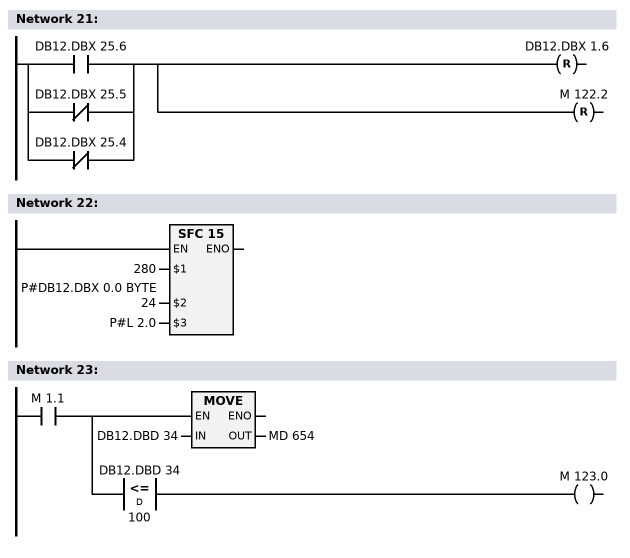
NETWORK
TITLE =
      O     DB12.DBX 25.6;
      ON    DB12.DBX 25.5;
      ON    DB12.DBX 25.4;
      R     DB12.DBX 1.6;
      R     M 122.2;
NETWORK
TITLE =
      CALL  SFC 15 (
           $1                       := 280,
           $2                       := P#DB12.DBX 0.0 BYTE 24,
           $3                       := P#L 2.0);
      NOP   0;
NETWORK
TITLE =
      A     M 1.1;
      =     L 20.0;
      A     L 20.0;
      JNB   M019;
      L     DB12.DBD 34;
      T     MD 654;
M019: NOP   0;
      A     L 20.0;
      A(;
      L     DB12.DBD 34;
      L     100;
      <=D;
      );
      =     M 123.0;
END_FUNCTION

FUNCTION FC 50 : VOID
VERSION : 0.1
BEGIN
// (block stored without names or comments; labels and parameter names are numbered)
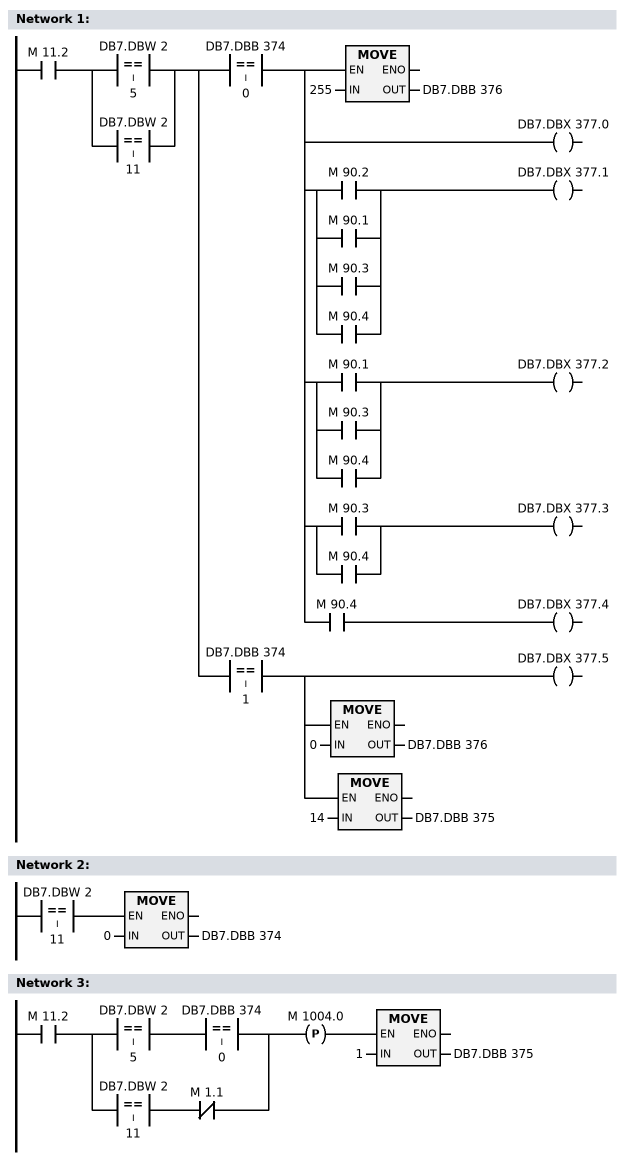
NETWORK
TITLE =
      A     M 11.2;
      A(;
      O(;
      L     DB7.DBW 2;
      L     5;
      ==I;
      );
      O(;
      L     DB7.DBW 2;
      L     11;
      ==I;
      );
      );
      =     L 8.0;
      A     L 8.0;
      A(;
      L     DB7.DBB 374;
      L     0;
      ==I;
      );
      =     L 8.1;
      A     L 8.1;
      JNB   M001;
      L     255;
      T     DB7.DBB 376;
M001: NOP   0;
      A     L 8.1;
      BLD   102;
      =     DB7.DBX 377.0;
      A     L 8.1;
      A(;
      O     M 90.2;
      O     M 90.1;
      O     M 90.3;
      O     M 90.4;
      );
      =     DB7.DBX 377.1;
      A     L 8.1;
      A(;
      O     M 90.1;
      O     M 90.3;
      O     M 90.4;
      );
      =     DB7.DBX 377.2;
      A     L 8.1;
      A(;
      O     M 90.3;
      O     M 90.4;
      );
      =     DB7.DBX 377.3;
      A     L 8.1;
      A     M 90.4;
      =     DB7.DBX 377.4;
      A     L 8.0;
      A(;
      L     DB7.DBB 374;
      L     1;
      ==I;
      );
      =     L 8.1;
      A     L 8.1;
      BLD   102;
      =     DB7.DBX 377.5;
      A     L 8.1;
      JNB   M002;
      L     0;
      T     DB7.DBB 376;
M002: NOP   0;
      A     L 8.1;
      JNB   M003;
      L     14;
      T     DB7.DBB 375;
M003: NOP   0;
NETWORK
TITLE =
      A(;
      L     DB7.DBW 2;
      L     11;
      ==I;
      );
      JNB   M004;
      L     0;
      T     DB7.DBB 374;
M004: NOP   0;
NETWORK
TITLE =
      A     M 11.2;
      A(;
      A(;
      L     DB7.DBW 2;
      L     5;
      ==I;
      );
      A(;
      L     DB7.DBB 374;
      L     0;
      ==I;
      );
      O;
      A(;
      L     DB7.DBW 2;
      L     11;
      ==I;
      );
      AN    M 1.1;
      );
      FP    M 1004.0;
      JNB   M005;
      L     1;
      T     DB7.DBB 375;
M005: NOP   0;
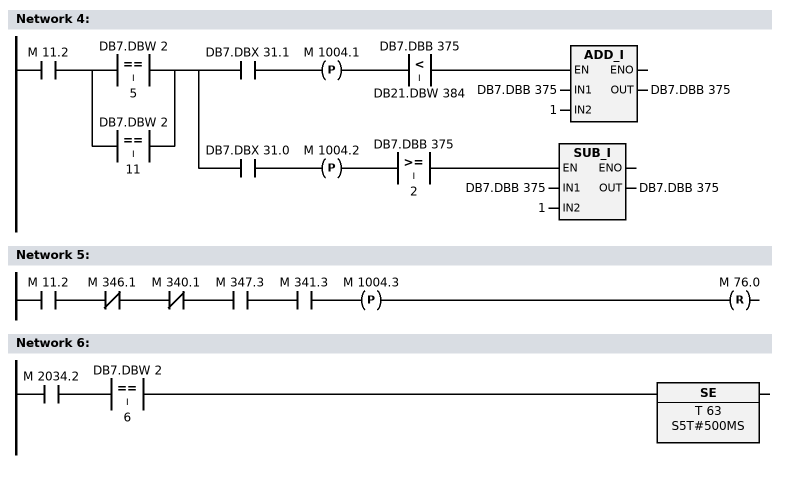
NETWORK
TITLE =
      A     M 11.2;
      A(;
      O(;
      L     DB7.DBW 2;
      L     5;
      ==I;
      );
      O(;
      L     DB7.DBW 2;
      L     11;
      ==I;
      );
      );
      =     L 8.0;
      A     L 8.0;
      A     DB7.DBX 31.1;
      FP    M 1004.1;
      A(;
      L     DB7.DBB 375;
      L     DB21.DBW 384;
      <I;
      );
      JNB   M006;
      L     DB7.DBB 375;
      L     1;
      +I;
      T     DB7.DBB 375;
M006: NOP   0;
      A     L 8.0;
      A     DB7.DBX 31.0;
      FP    M 1004.2;
      A(;
      L     DB7.DBB 375;
      L     2;
      >=I;
      );
      JNB   M007;
      L     DB7.DBB 375;
      L     1;
      -I;
      T     DB7.DBB 375;
M007: NOP   0;
NETWORK
TITLE =
      A     M 11.2;
      AN    M 346.1;
      AN    M 340.1;
      A     M 347.3;
      A     M 341.3;
      FP    M 1004.3;
      R     M 76.0;
NETWORK
TITLE =
      A     M 2034.2;
      A(;
      L     DB7.DBW 2;
      L     6;
      ==I;
      );
      L     S5T#500MS;
      SE    T 63;
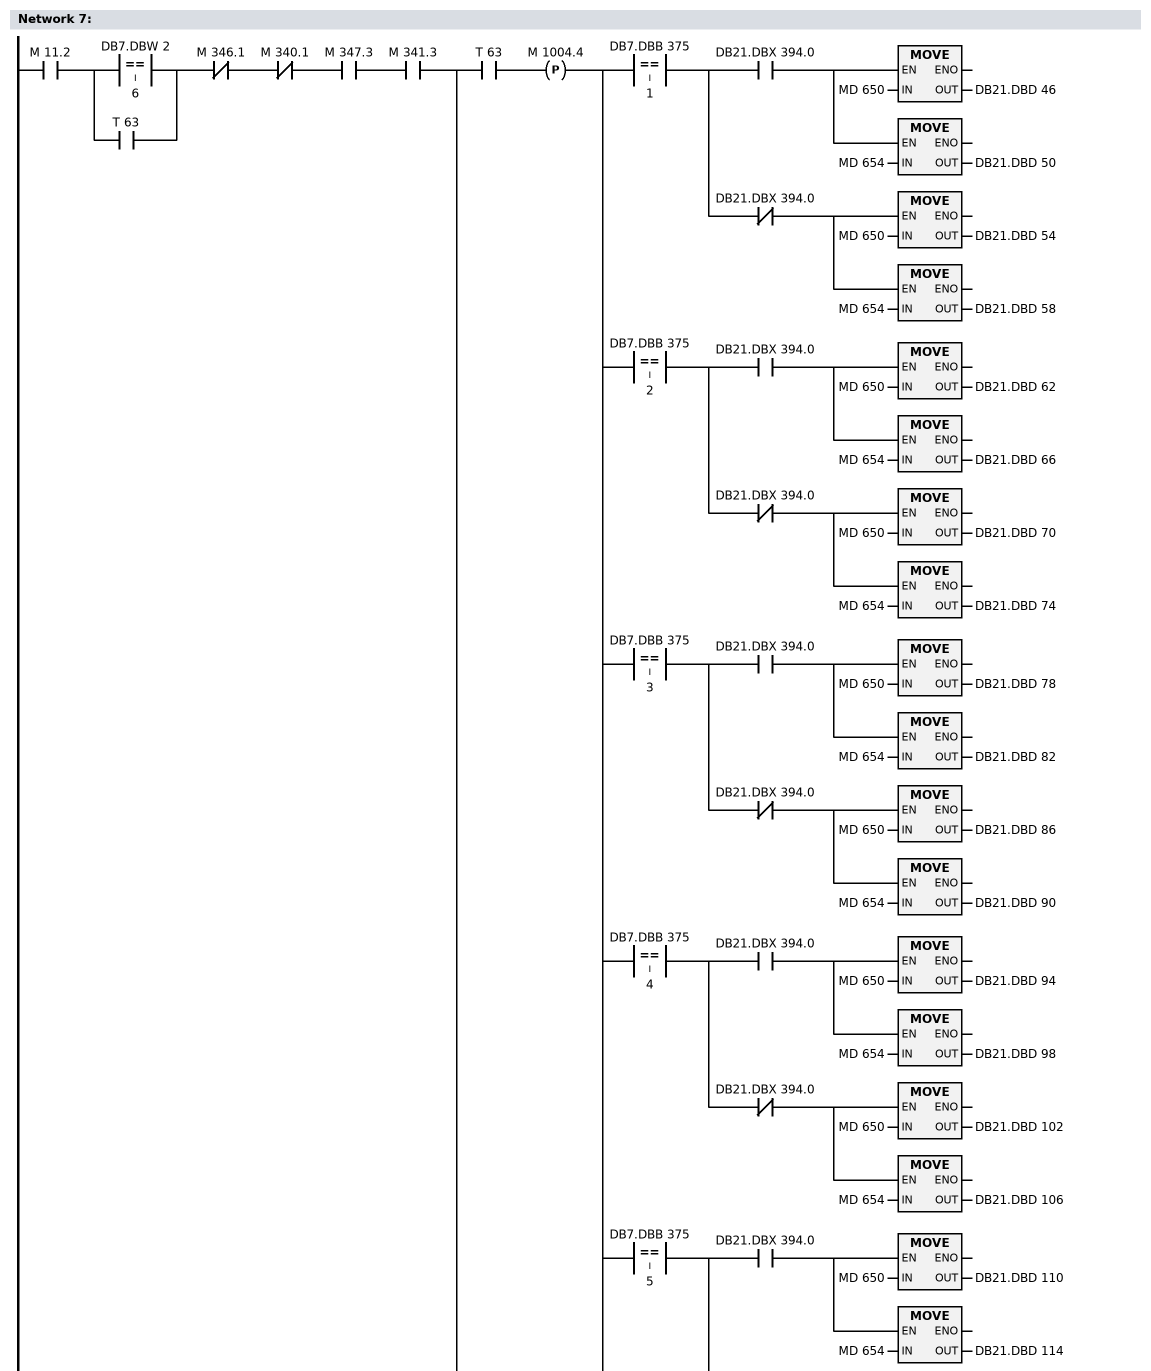
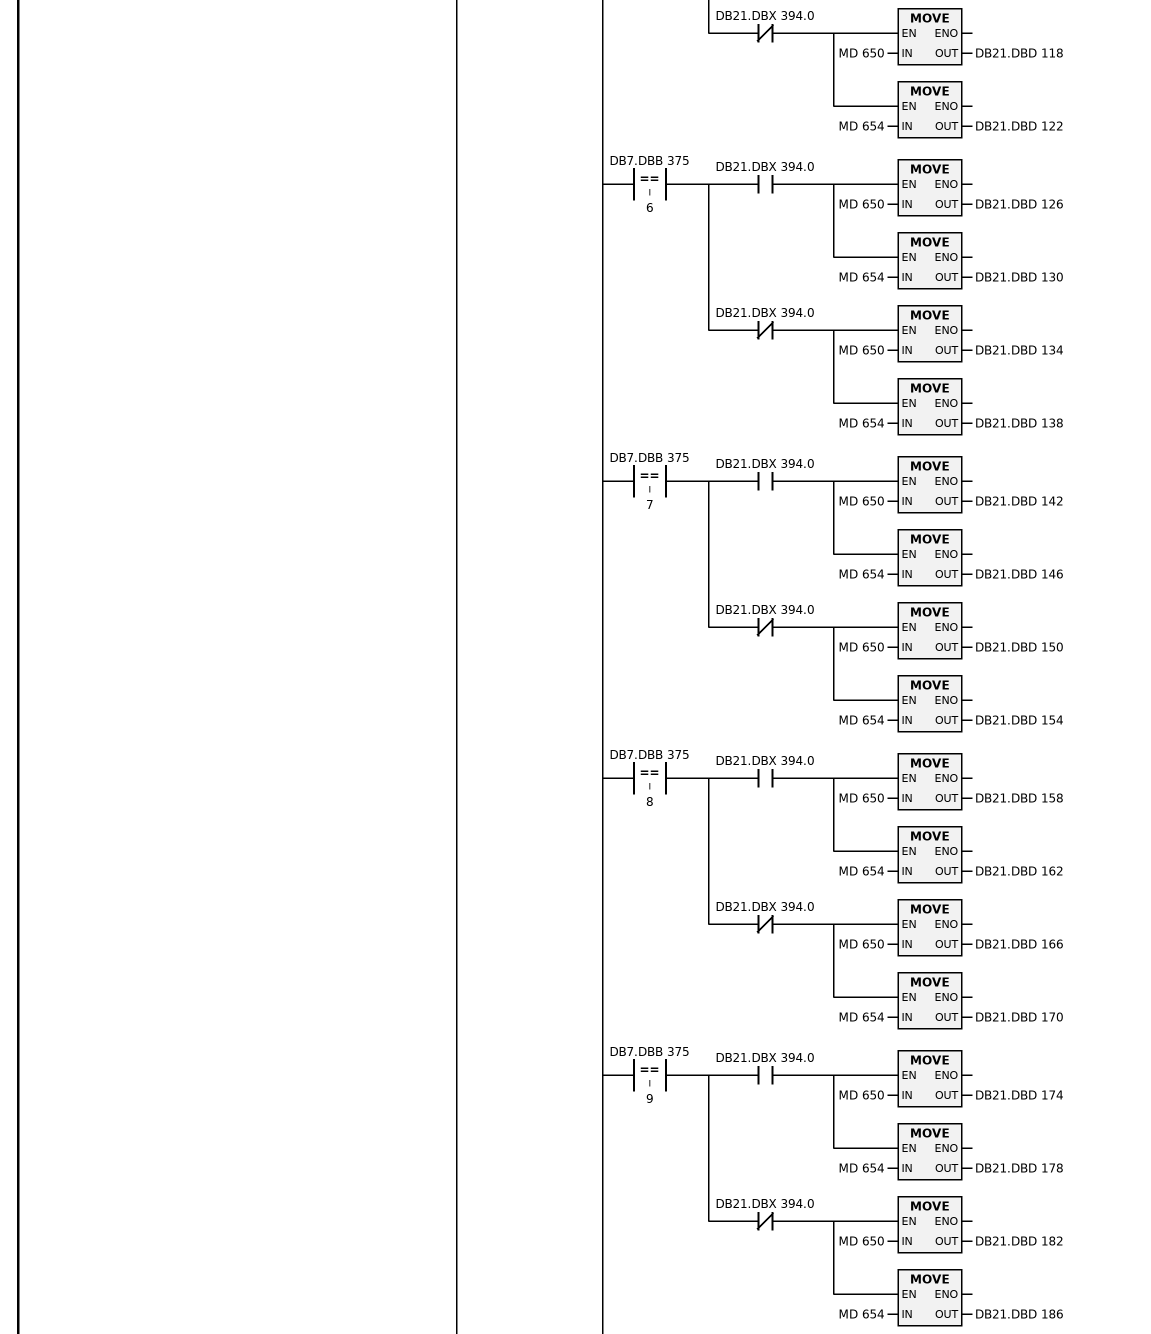
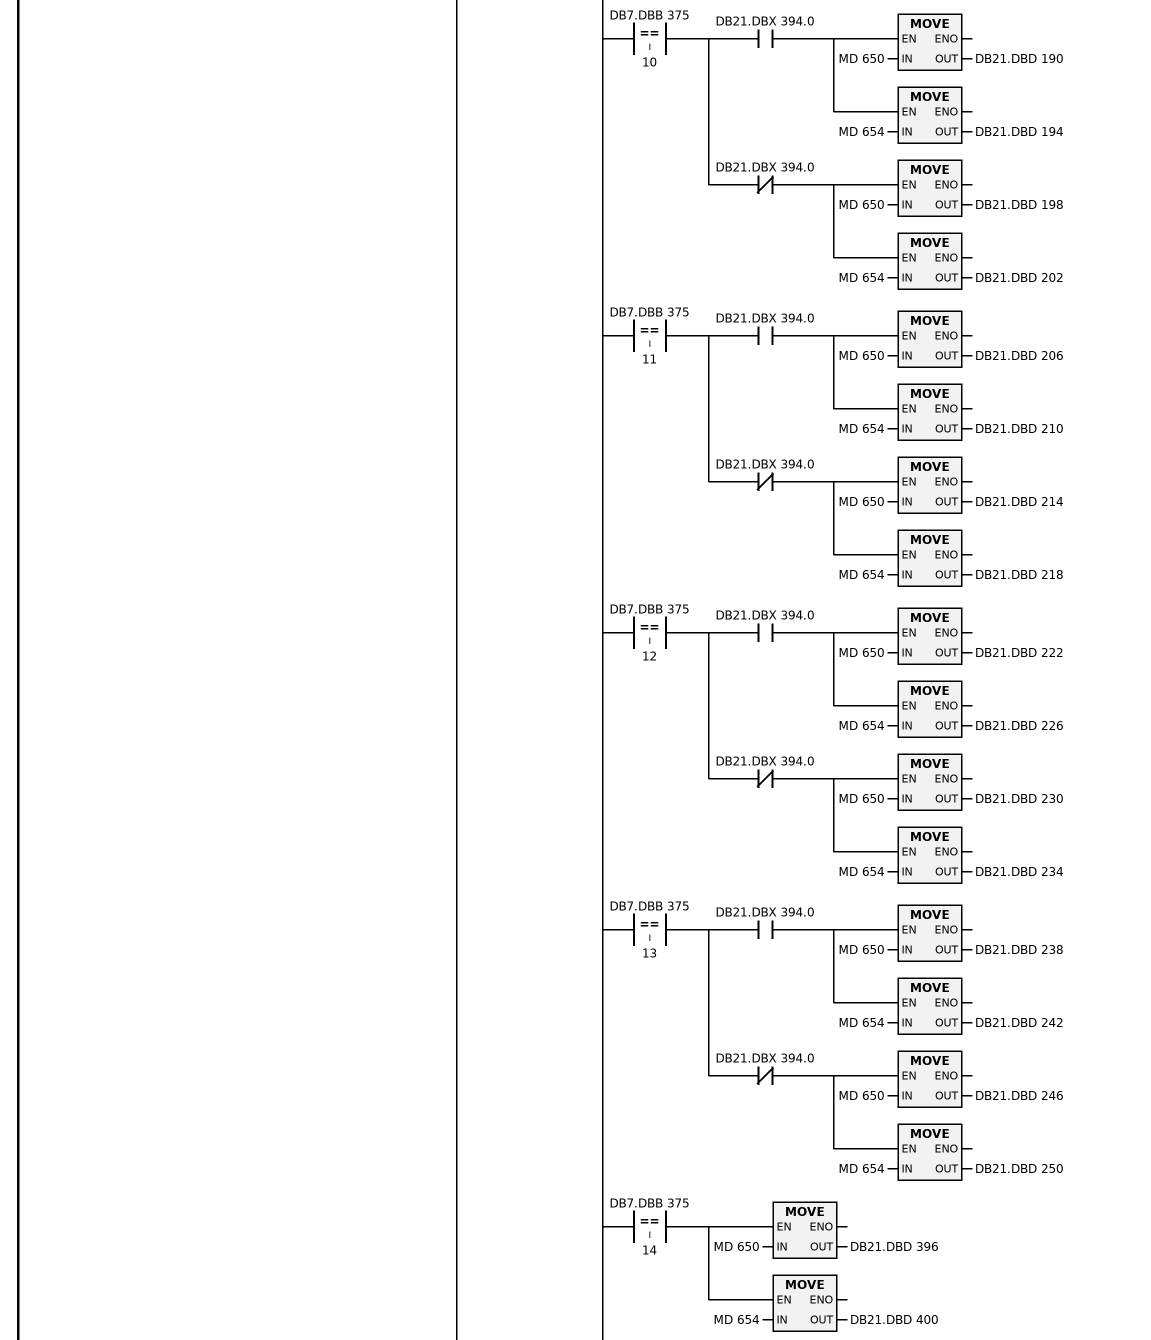
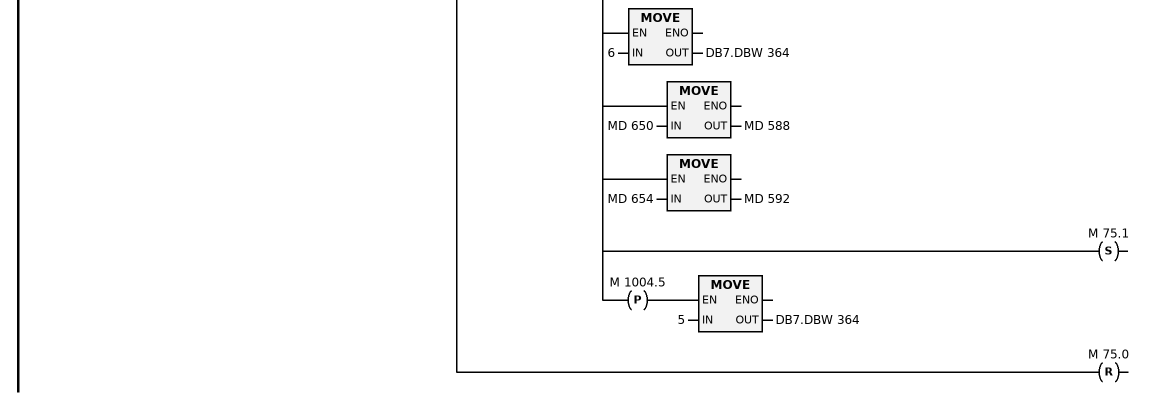
NETWORK
TITLE =
      A     M 11.2;
      A(;
      O(;
      L     DB7.DBW 2;
      L     6;
      ==I;
      );
      O     T 63;
      );
      AN    M 346.1;
      AN    M 340.1;
      A     M 347.3;
      A     M 341.3;
      =     L 8.0;
      A     L 8.0;
      A     T 63;
      FP    M 1004.4;
      =     L 8.1;
      A     L 8.1;
      A(;
      L     DB7.DBB 375;
      L     1;
      ==I;
      );
      =     L 8.2;
      A     L 8.2;
      A     DB21.DBX 394.0;
      =     L 8.3;
      A     L 8.3;
      JNB   M008;
      L     MD 650;
      T     DB21.DBD 46;
M008: NOP   0;
      A     L 8.3;
      JNB   M009;
      L     MD 654;
      T     DB21.DBD 50;
M009: NOP   0;
      A     L 8.2;
      AN    DB21.DBX 394.0;
      =     L 8.3;
      A     L 8.3;
      JNB   M010;
      L     MD 650;
      T     DB21.DBD 54;
M010: NOP   0;
      A     L 8.3;
      JNB   M011;
      L     MD 654;
      T     DB21.DBD 58;
M011: NOP   0;
      A     L 8.1;
      A(;
      L     DB7.DBB 375;
      L     2;
      ==I;
      );
      =     L 8.2;
      A     L 8.2;
      A     DB21.DBX 394.0;
      =     L 8.3;
      A     L 8.3;
      JNB   M012;
      L     MD 650;
      T     DB21.DBD 62;
M012: NOP   0;
      A     L 8.3;
      JNB   M013;
      L     MD 654;
      T     DB21.DBD 66;
M013: NOP   0;
      A     L 8.2;
      AN    DB21.DBX 394.0;
      =     L 8.3;
      A     L 8.3;
      JNB   M014;
      L     MD 650;
      T     DB21.DBD 70;
M014: NOP   0;
      A     L 8.3;
      JNB   M015;
      L     MD 654;
      T     DB21.DBD 74;
M015: NOP   0;
      A     L 8.1;
      A(;
      L     DB7.DBB 375;
      L     3;
      ==I;
      );
      =     L 8.2;
      A     L 8.2;
      A     DB21.DBX 394.0;
      =     L 8.3;
      A     L 8.3;
      JNB   M016;
      L     MD 650;
      T     DB21.DBD 78;
M016: NOP   0;
      A     L 8.3;
      JNB   M017;
      L     MD 654;
      T     DB21.DBD 82;
M017: NOP   0;
      A     L 8.2;
      AN    DB21.DBX 394.0;
      =     L 8.3;
      A     L 8.3;
      JNB   M018;
      L     MD 650;
      T     DB21.DBD 86;
M018: NOP   0;
      A     L 8.3;
      JNB   M019;
      L     MD 654;
      T     DB21.DBD 90;
M019: NOP   0;
      A     L 8.1;
      A(;
      L     DB7.DBB 375;
      L     4;
      ==I;
      );
      =     L 8.2;
      A     L 8.2;
      A     DB21.DBX 394.0;
      =     L 8.3;
      A     L 8.3;
      JNB   M020;
      L     MD 650;
      T     DB21.DBD 94;
M020: NOP   0;
      A     L 8.3;
      JNB   M021;
      L     MD 654;
      T     DB21.DBD 98;
M021: NOP   0;
      A     L 8.2;
      AN    DB21.DBX 394.0;
      =     L 8.3;
      A     L 8.3;
      JNB   M022;
      L     MD 650;
      T     DB21.DBD 102;
M022: NOP   0;
      A     L 8.3;
      JNB   M023;
      L     MD 654;
      T     DB21.DBD 106;
M023: NOP   0;
      A     L 8.1;
      A(;
      L     DB7.DBB 375;
      L     5;
      ==I;
      );
      =     L 8.2;
      A     L 8.2;
      A     DB21.DBX 394.0;
      =     L 8.3;
      A     L 8.3;
      JNB   M024;
      L     MD 650;
      T     DB21.DBD 110;
M024: NOP   0;
      A     L 8.3;
      JNB   M025;
      L     MD 654;
      T     DB21.DBD 114;
M025: NOP   0;
      A     L 8.2;
      AN    DB21.DBX 394.0;
      =     L 8.3;
      A     L 8.3;
      JNB   M026;
      L     MD 650;
      T     DB21.DBD 118;
M026: NOP   0;
      A     L 8.3;
      JNB   M027;
      L     MD 654;
      T     DB21.DBD 122;
M027: NOP   0;
      A     L 8.1;
      A(;
      L     DB7.DBB 375;
      L     6;
      ==I;
      );
      =     L 8.2;
      A     L 8.2;
      A     DB21.DBX 394.0;
      =     L 8.3;
      A     L 8.3;
      JNB   M028;
      L     MD 650;
      T     DB21.DBD 126;
M028: NOP   0;
      A     L 8.3;
      JNB   M029;
      L     MD 654;
      T     DB21.DBD 130;
M029: NOP   0;
      A     L 8.2;
      AN    DB21.DBX 394.0;
      =     L 8.3;
      A     L 8.3;
      JNB   M030;
      L     MD 650;
      T     DB21.DBD 134;
M030: NOP   0;
      A     L 8.3;
      JNB   M031;
      L     MD 654;
      T     DB21.DBD 138;
M031: NOP   0;
      A     L 8.1;
      A(;
      L     DB7.DBB 375;
      L     7;
      ==I;
      );
      =     L 8.2;
      A     L 8.2;
      A     DB21.DBX 394.0;
      =     L 8.3;
      A     L 8.3;
      JNB   M032;
      L     MD 650;
      T     DB21.DBD 142;
M032: NOP   0;
      A     L 8.3;
      JNB   M033;
      L     MD 654;
      T     DB21.DBD 146;
M033: NOP   0;
      A     L 8.2;
      AN    DB21.DBX 394.0;
      =     L 8.3;
      A     L 8.3;
      JNB   M034;
      L     MD 650;
      T     DB21.DBD 150;
M034: NOP   0;
      A     L 8.3;
      JNB   M035;
      L     MD 654;
      T     DB21.DBD 154;
M035: NOP   0;
      A     L 8.1;
      A(;
      L     DB7.DBB 375;
      L     8;
      ==I;
      );
      =     L 8.2;
      A     L 8.2;
      A     DB21.DBX 394.0;
      =     L 8.3;
      A     L 8.3;
      JNB   M036;
      L     MD 650;
      T     DB21.DBD 158;
M036: NOP   0;
      A     L 8.3;
      JNB   M037;
      L     MD 654;
      T     DB21.DBD 162;
M037: NOP   0;
      A     L 8.2;
      AN    DB21.DBX 394.0;
      =     L 8.3;
      A     L 8.3;
      JNB   M038;
      L     MD 650;
      T     DB21.DBD 166;
M038: NOP   0;
      A     L 8.3;
      JNB   M039;
      L     MD 654;
      T     DB21.DBD 170;
M039: NOP   0;
      A     L 8.1;
      A(;
      L     DB7.DBB 375;
      L     9;
      ==I;
      );
      =     L 8.2;
      A     L 8.2;
      A     DB21.DBX 394.0;
      =     L 8.3;
      A     L 8.3;
      JNB   M040;
      L     MD 650;
      T     DB21.DBD 174;
M040: NOP   0;
      A     L 8.3;
      JNB   M041;
      L     MD 654;
      T     DB21.DBD 178;
M041: NOP   0;
      A     L 8.2;
      AN    DB21.DBX 394.0;
      =     L 8.3;
      A     L 8.3;
      JNB   M042;
      L     MD 650;
      T     DB21.DBD 182;
M042: NOP   0;
      A     L 8.3;
      JNB   M043;
      L     MD 654;
      T     DB21.DBD 186;
M043: NOP   0;
      A     L 8.1;
      A(;
      L     DB7.DBB 375;
      L     10;
      ==I;
      );
      =     L 8.2;
      A     L 8.2;
      A     DB21.DBX 394.0;
      =     L 8.3;
      A     L 8.3;
      JNB   M044;
      L     MD 650;
      T     DB21.DBD 190;
M044: NOP   0;
      A     L 8.3;
      JNB   M045;
      L     MD 654;
      T     DB21.DBD 194;
M045: NOP   0;
      A     L 8.2;
      AN    DB21.DBX 394.0;
      =     L 8.3;
      A     L 8.3;
      JNB   M046;
      L     MD 650;
      T     DB21.DBD 198;
M046: NOP   0;
      A     L 8.3;
      JNB   M047;
      L     MD 654;
      T     DB21.DBD 202;
M047: NOP   0;
      A     L 8.1;
      A(;
      L     DB7.DBB 375;
      L     11;
      ==I;
      );
      =     L 8.2;
      A     L 8.2;
      A     DB21.DBX 394.0;
      =     L 8.3;
      A     L 8.3;
      JNB   M048;
      L     MD 650;
      T     DB21.DBD 206;
M048: NOP   0;
      A     L 8.3;
      JNB   M049;
      L     MD 654;
      T     DB21.DBD 210;
M049: NOP   0;
      A     L 8.2;
      AN    DB21.DBX 394.0;
      =     L 8.3;
      A     L 8.3;
      JNB   M050;
      L     MD 650;
      T     DB21.DBD 214;
M050: NOP   0;
      A     L 8.3;
      JNB   M051;
      L     MD 654;
      T     DB21.DBD 218;
M051: NOP   0;
      A     L 8.1;
      A(;
      L     DB7.DBB 375;
      L     12;
      ==I;
      );
      =     L 8.2;
      A     L 8.2;
      A     DB21.DBX 394.0;
      =     L 8.3;
      A     L 8.3;
      JNB   M052;
      L     MD 650;
      T     DB21.DBD 222;
M052: NOP   0;
      A     L 8.3;
      JNB   M053;
      L     MD 654;
      T     DB21.DBD 226;
M053: NOP   0;
      A     L 8.2;
      AN    DB21.DBX 394.0;
      =     L 8.3;
      A     L 8.3;
      JNB   M054;
      L     MD 650;
      T     DB21.DBD 230;
M054: NOP   0;
      A     L 8.3;
      JNB   M055;
      L     MD 654;
      T     DB21.DBD 234;
M055: NOP   0;
      A     L 8.1;
      A(;
      L     DB7.DBB 375;
      L     13;
      ==I;
      );
      =     L 8.2;
      A     L 8.2;
      A     DB21.DBX 394.0;
      =     L 8.3;
      A     L 8.3;
      JNB   M056;
      L     MD 650;
      T     DB21.DBD 238;
M056: NOP   0;
      A     L 8.3;
      JNB   M057;
      L     MD 654;
      T     DB21.DBD 242;
M057: NOP   0;
      A     L 8.2;
      AN    DB21.DBX 394.0;
      =     L 8.3;
      A     L 8.3;
      JNB   M058;
      L     MD 650;
      T     DB21.DBD 246;
M058: NOP   0;
      A     L 8.3;
      JNB   M059;
      L     MD 654;
      T     DB21.DBD 250;
M059: NOP   0;
      A     L 8.1;
      A(;
      L     DB7.DBB 375;
      L     14;
      ==I;
      );
      =     L 8.2;
      A     L 8.2;
      JNB   M060;
      L     MD 650;
      T     DB21.DBD 396;
M060: NOP   0;
      A     L 8.2;
      JNB   M061;
      L     MD 654;
      T     DB21.DBD 400;
M061: NOP   0;
      A     L 8.1;
      JNB   M062;
      L     6;
      T     DB7.DBW 364;
M062: NOP   0;
      A     L 8.1;
      JNB   M063;
      L     MD 650;
      T     MD 588;
M063: NOP   0;
      A     L 8.1;
      JNB   M064;
      L     MD 654;
      T     MD 592;
M064: NOP   0;
      A     L 8.1;
      BLD   102;
      S     M 75.1;
      A     L 8.1;
      FP    M 1004.5;
      JNB   M065;
      L     5;
      T     DB7.DBW 364;
M065: NOP   0;
      A     L 8.0;
      BLD   102;
      R     M 75.0;
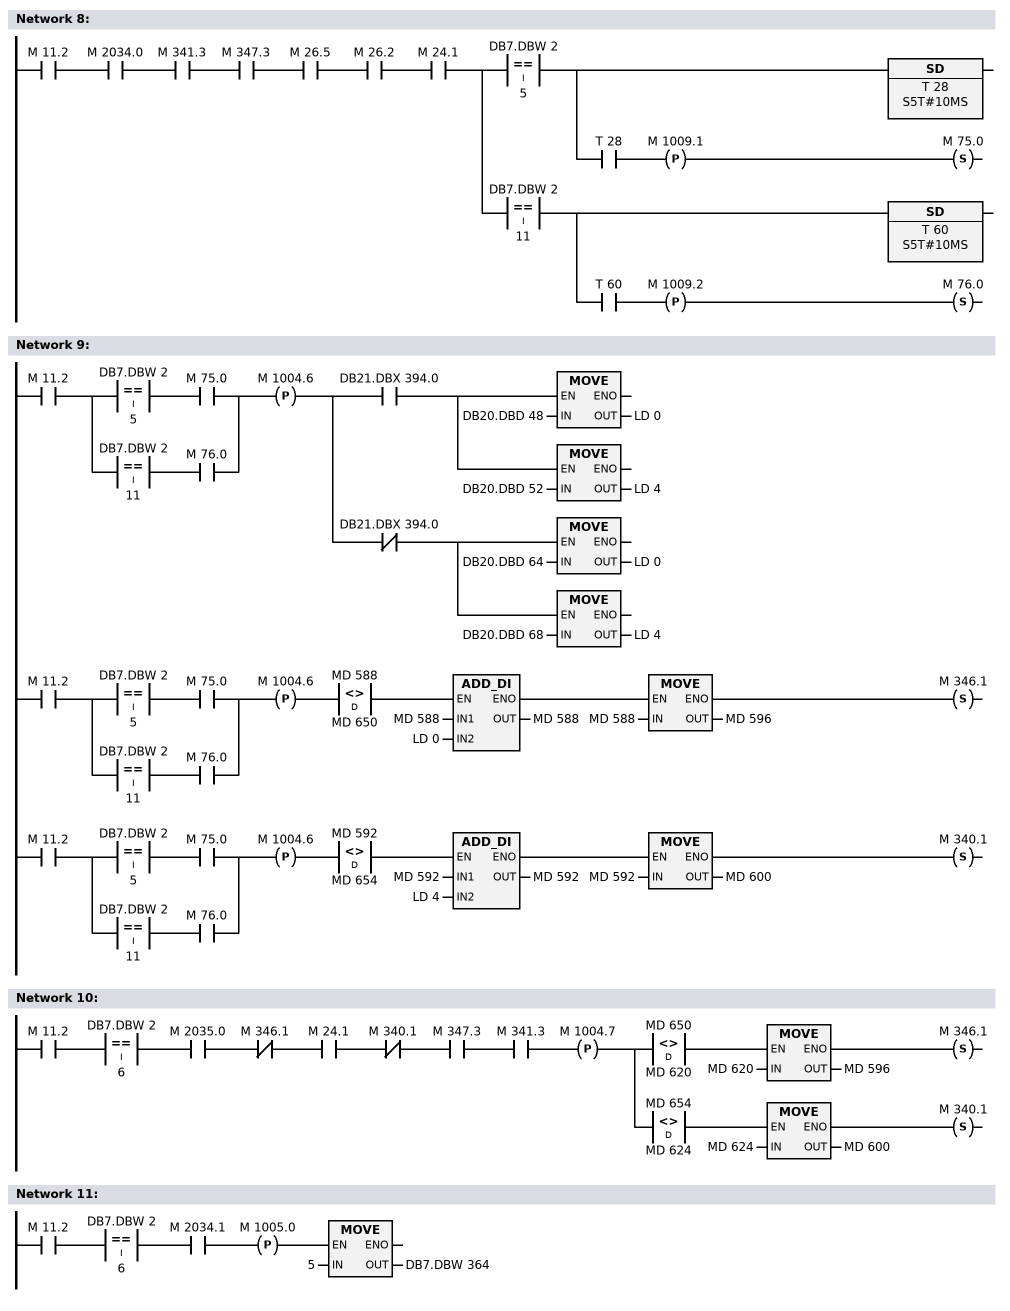
NETWORK
TITLE =
      A     M 11.2;
      A     M 2034.0;
      A     M 341.3;
      A     M 347.3;
      A     M 26.5;
      A     M 26.2;
      A     M 24.1;
      =     L 8.0;
      A     L 8.0;
      A(;
      L     DB7.DBW 2;
      L     5;
      ==I;
      );
      =     L 8.1;
      A     L 8.1;
      BLD   102;
      L     S5T#10MS;
      SD    T 28;
      A     L 8.1;
      A     T 28;
      FP    M 1009.1;
      S     M 75.0;
      A     L 8.0;
      A(;
      L     DB7.DBW 2;
      L     11;
      ==I;
      );
      =     L 8.1;
      A     L 8.1;
      BLD   102;
      L     S5T#10MS;
      SD    T 60;
      A     L 8.1;
      A     T 60;
      FP    M 1009.2;
      S     M 76.0;
NETWORK
TITLE =
      A     M 11.2;
      A(;
      A(;
      L     DB7.DBW 2;
      L     5;
      ==I;
      );
      A     M 75.0;
      O;
      A(;
      L     DB7.DBW 2;
      L     11;
      ==I;
      );
      A     M 76.0;
      );
      FP    M 1004.6;
      =     L 8.0;
      A     L 8.0;
      A     DB21.DBX 394.0;
      =     L 8.1;
      A     L 8.1;
      JNB   M066;
      L     DB20.DBD 48;
      T     LD 0;
M066: NOP   0;
      A     L 8.1;
      JNB   M067;
      L     DB20.DBD 52;
      T     LD 4;
M067: NOP   0;
      A     L 8.0;
      AN    DB21.DBX 394.0;
      =     L 8.1;
      A     L 8.1;
      JNB   M068;
      L     DB20.DBD 64;
      T     LD 0;
M068: NOP   0;
      A     L 8.1;
      JNB   M069;
      L     DB20.DBD 68;
      T     LD 4;
M069: NOP   0;
      A(;
      A     L 8.0;
      A(;
      L     MD 588;
      L     MD 650;
      <>D;
      );
      JNB   M070;
      L     MD 588;
      L     LD 0;
      +D;
      T     MD 588;
      AN    OV;
      SAVE;
      CLR;
M070: A     BR;
      );
      JNB   M071;
      L     MD 588;
      T     MD 596;
      SET;
      SAVE;
      CLR;
M071: A     BR;
      S     M 346.1;
      A(;
      A     L 8.0;
      A(;
      L     MD 592;
      L     MD 654;
      <>D;
      );
      JNB   M072;
      L     MD 592;
      L     LD 4;
      +D;
      T     MD 592;
      AN    OV;
      SAVE;
      CLR;
M072: A     BR;
      );
      JNB   M073;
      L     MD 592;
      T     MD 600;
      SET;
      SAVE;
      CLR;
M073: A     BR;
      S     M 340.1;
NETWORK
TITLE =
      A     M 11.2;
      A(;
      L     DB7.DBW 2;
      L     6;
      ==I;
      );
      A     M 2035.0;
      AN    M 346.1;
      A     M 24.1;
      AN    M 340.1;
      A     M 347.3;
      A     M 341.3;
      FP    M 1004.7;
      =     L 8.0;
      A     L 8.0;
      A(;
      L     MD 650;
      L     MD 620;
      <>D;
      );
      JNB   M074;
      L     MD 620;
      T     MD 596;
      SET;
      SAVE;
      CLR;
M074: A     BR;
      S     M 346.1;
      A     L 8.0;
      A(;
      L     MD 654;
      L     MD 624;
      <>D;
      );
      JNB   M075;
      L     MD 624;
      T     MD 600;
      SET;
      SAVE;
      CLR;
M075: A     BR;
      S     M 340.1;
NETWORK
TITLE =
      A     M 11.2;
      A(;
      L     DB7.DBW 2;
      L     6;
      ==I;
      );
      A     M 2034.1;
      FP    M 1005.0;
      JNB   M076;
      L     5;
      T     DB7.DBW 364;
M076: NOP   0;
END_FUNCTION

FUNCTION FC 51 : VOID
VERSION : 0.1
BEGIN
// (block stored without names or comments; labels and parameter names are numbered)
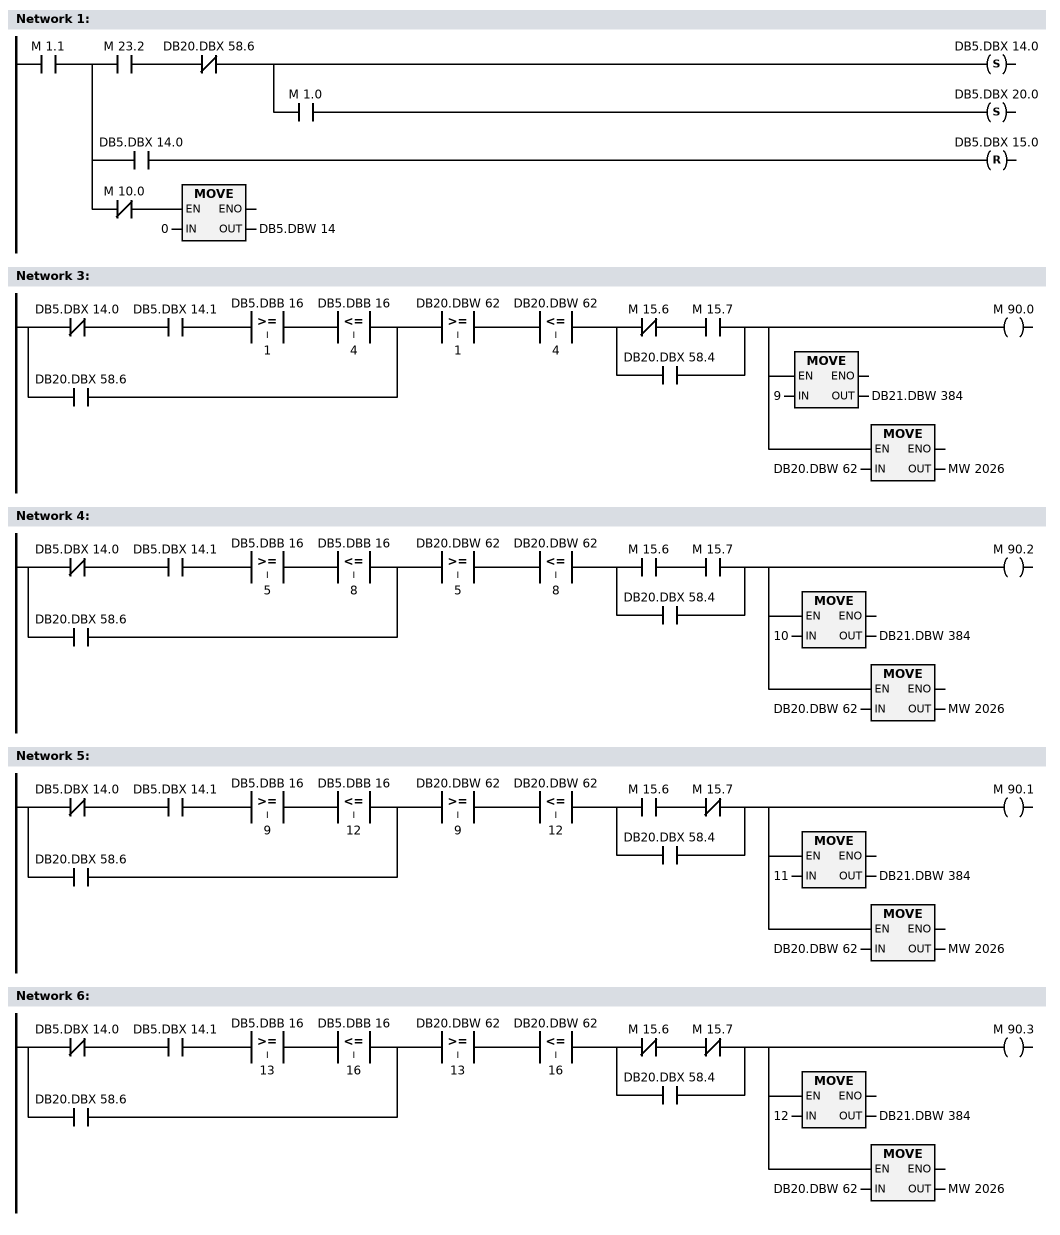
NETWORK
TITLE =
      A     M 1.1;
      =     L 0.0;
      A     L 0.0;
      A     M 23.2;
      AN    DB20.DBX 58.6;
      =     L 0.1;
      A     L 0.1;
      BLD   102;
      S     DB5.DBX 14.0;
      A     L 0.1;
      A     M 1.0;
      S     DB5.DBX 20.0;
      A     L 0.0;
      A     DB5.DBX 14.0;
      R     DB5.DBX 15.0;
      A     L 0.0;
      AN    M 10.0;
      JNB   M001;
      L     0;
      T     DB5.DBW 14;
M001: NOP   0;
NETWORK
TITLE =
NETWORK
TITLE =
      A(;
      AN    DB5.DBX 14.0;
      A     DB5.DBX 14.1;
      A(;
      L     DB5.DBB 16;
      L     1;
      >=I;
      );
      A(;
      L     DB5.DBB 16;
      L     4;
      <=I;
      );
      O     DB20.DBX 58.6;
      );
      A(;
      L     DB20.DBW 62;
      L     1;
      >=I;
      );
      A(;
      L     DB20.DBW 62;
      L     4;
      <=I;
      );
      A(;
      AN    M 15.6;
      A     M 15.7;
      O     DB20.DBX 58.4;
      );
      =     L 0.0;
      A     L 0.0;
      BLD   102;
      =     M 90.0;
      A     L 0.0;
      JNB   M002;
      L     9;
      T     DB21.DBW 384;
M002: NOP   0;
      A     L 0.0;
      JNB   M003;
      L     DB20.DBW 62;
      T     MW 2026;
M003: NOP   0;
NETWORK
TITLE =
      A(;
      AN    DB5.DBX 14.0;
      A     DB5.DBX 14.1;
      A(;
      L     DB5.DBB 16;
      L     5;
      >=I;
      );
      A(;
      L     DB5.DBB 16;
      L     8;
      <=I;
      );
      O     DB20.DBX 58.6;
      );
      A(;
      L     DB20.DBW 62;
      L     5;
      >=I;
      );
      A(;
      L     DB20.DBW 62;
      L     8;
      <=I;
      );
      A(;
      A     M 15.6;
      A     M 15.7;
      O     DB20.DBX 58.4;
      );
      =     L 0.0;
      A     L 0.0;
      BLD   102;
      =     M 90.2;
      A     L 0.0;
      JNB   M004;
      L     10;
      T     DB21.DBW 384;
M004: NOP   0;
      A     L 0.0;
      JNB   M005;
      L     DB20.DBW 62;
      T     MW 2026;
M005: NOP   0;
NETWORK
TITLE =
      A(;
      AN    DB5.DBX 14.0;
      A     DB5.DBX 14.1;
      A(;
      L     DB5.DBB 16;
      L     9;
      >=I;
      );
      A(;
      L     DB5.DBB 16;
      L     12;
      <=I;
      );
      O     DB20.DBX 58.6;
      );
      A(;
      L     DB20.DBW 62;
      L     9;
      >=I;
      );
      A(;
      L     DB20.DBW 62;
      L     12;
      <=I;
      );
      A(;
      A     M 15.6;
      AN    M 15.7;
      O     DB20.DBX 58.4;
      );
      =     L 0.0;
      A     L 0.0;
      BLD   102;
      =     M 90.1;
      A     L 0.0;
      JNB   M006;
      L     11;
      T     DB21.DBW 384;
M006: NOP   0;
      A     L 0.0;
      JNB   M007;
      L     DB20.DBW 62;
      T     MW 2026;
M007: NOP   0;
NETWORK
TITLE =
      A(;
      AN    DB5.DBX 14.0;
      A     DB5.DBX 14.1;
      A(;
      L     DB5.DBB 16;
      L     13;
      >=I;
      );
      A(;
      L     DB5.DBB 16;
      L     16;
      <=I;
      );
      O     DB20.DBX 58.6;
      );
      A(;
      L     DB20.DBW 62;
      L     13;
      >=I;
      );
      A(;
      L     DB20.DBW 62;
      L     16;
      <=I;
      );
      A(;
      AN    M 15.6;
      AN    M 15.7;
      O     DB20.DBX 58.4;
      );
      =     L 0.0;
      A     L 0.0;
      BLD   102;
      =     M 90.3;
      A     L 0.0;
      JNB   M008;
      L     12;
      T     DB21.DBW 384;
M008: NOP   0;
      A     L 0.0;
      JNB   M009;
      L     DB20.DBW 62;
      T     MW 2026;
M009: NOP   0;
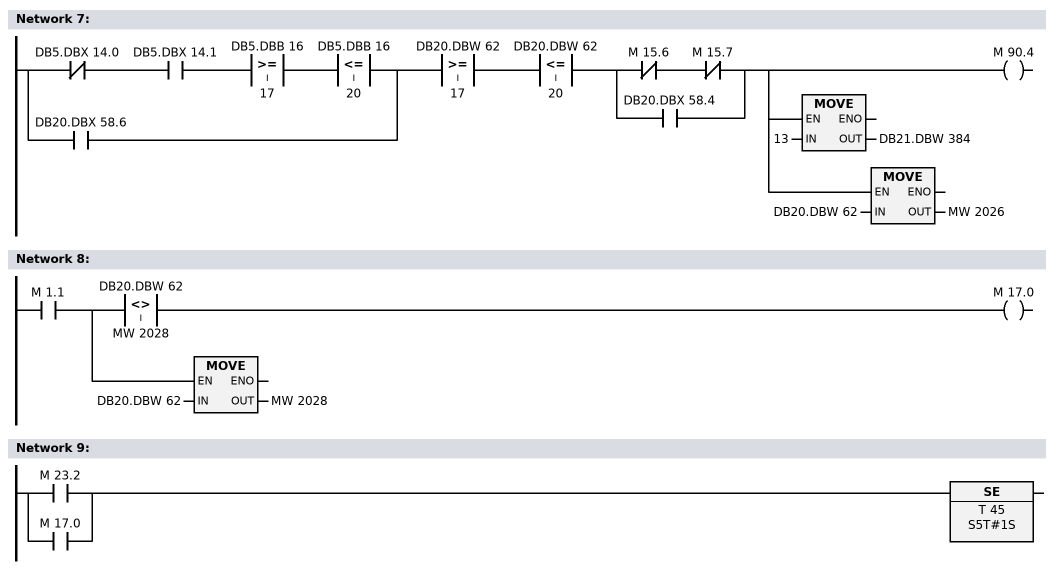
NETWORK
TITLE =
      A(;
      AN    DB5.DBX 14.0;
      A     DB5.DBX 14.1;
      A(;
      L     DB5.DBB 16;
      L     17;
      >=I;
      );
      A(;
      L     DB5.DBB 16;
      L     20;
      <=I;
      );
      O     DB20.DBX 58.6;
      );
      A(;
      L     DB20.DBW 62;
      L     17;
      >=I;
      );
      A(;
      L     DB20.DBW 62;
      L     20;
      <=I;
      );
      A(;
      AN    M 15.6;
      AN    M 15.7;
      O     DB20.DBX 58.4;
      );
      =     L 0.0;
      A     L 0.0;
      BLD   102;
      =     M 90.4;
      A     L 0.0;
      JNB   M010;
      L     13;
      T     DB21.DBW 384;
M010: NOP   0;
      A     L 0.0;
      JNB   M011;
      L     DB20.DBW 62;
      T     MW 2026;
M011: NOP   0;
NETWORK
TITLE =
      A     M 1.1;
      =     L 0.0;
      A     L 0.0;
      A(;
      L     DB20.DBW 62;
      L     MW 2028;
      <>I;
      );
      =     M 17.0;
      A     L 0.0;
      JNB   M012;
      L     DB20.DBW 62;
      T     MW 2028;
M012: NOP   0;
NETWORK
TITLE =
      O     M 23.2;
      O     M 17.0;
      L     S5T#1S;
      SE    T 45;
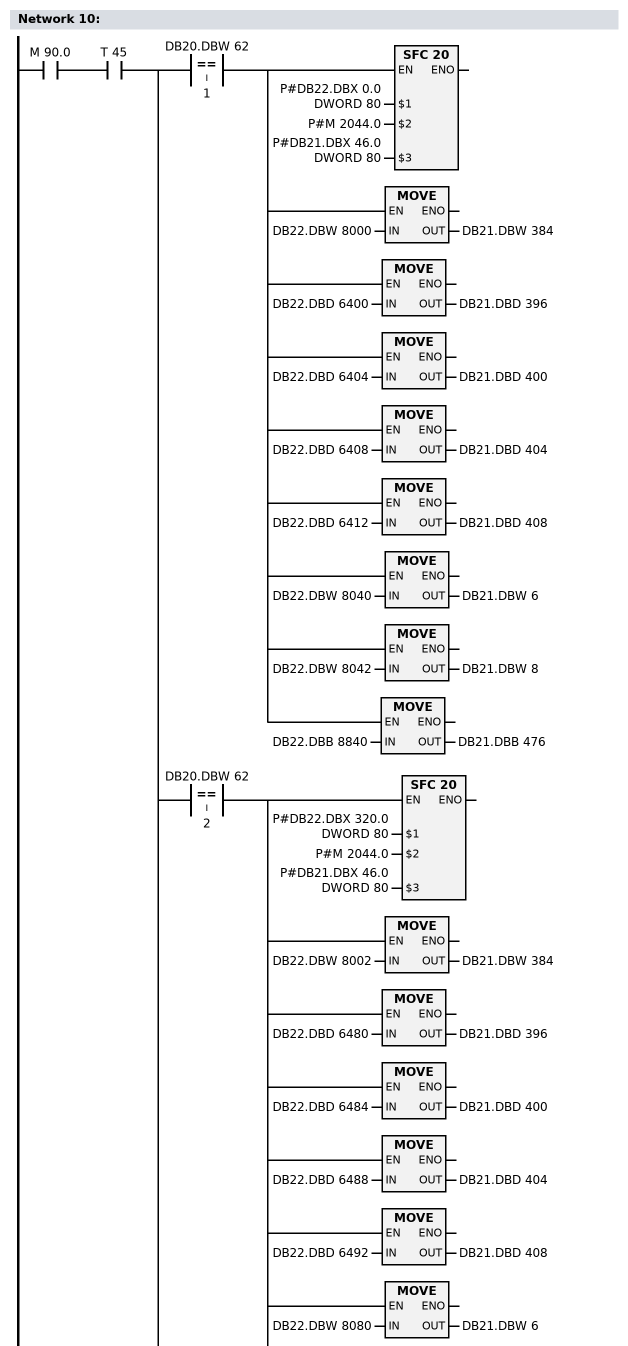
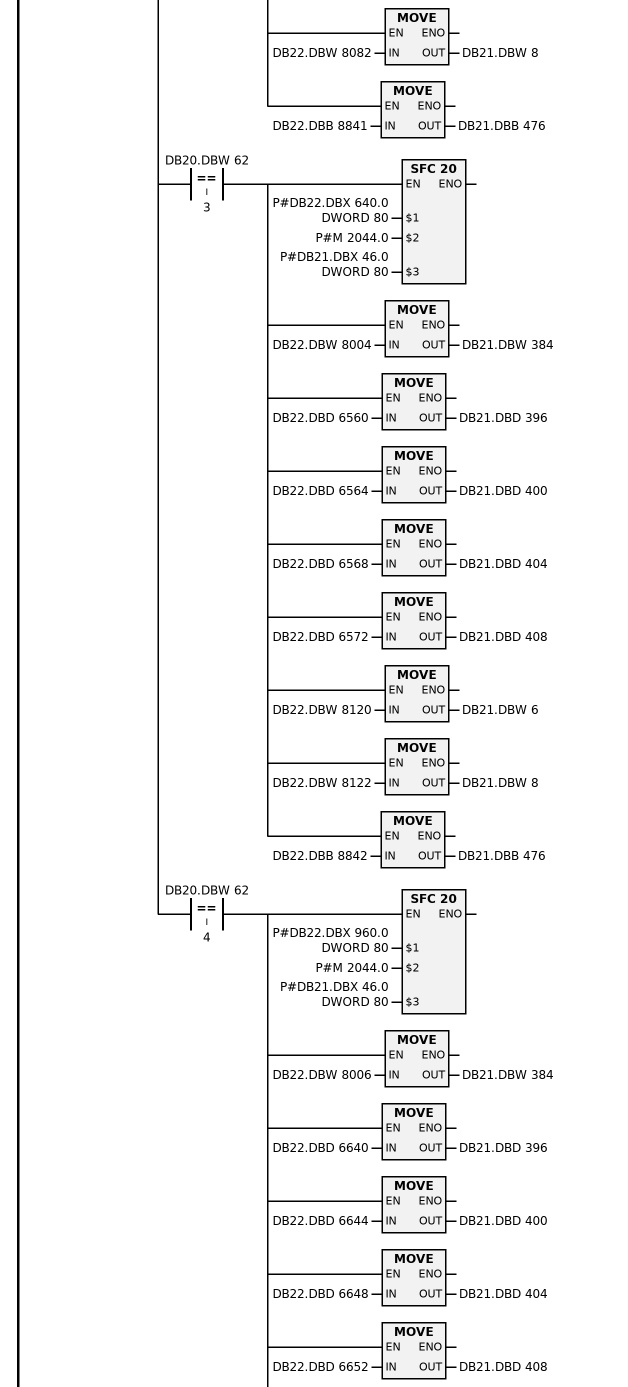
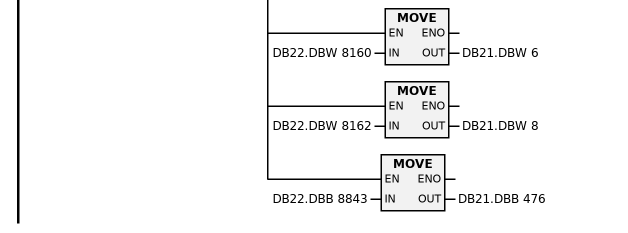
NETWORK
TITLE =
      A     M 90.0;
      A     T 45;
      =     L 0.0;
      A     L 0.0;
      A(;
      L     DB20.DBW 62;
      L     1;
      ==I;
      );
      =     L 0.1;
      A     L 0.1;
      JNB   M013;
      CALL  SFC 20 (
           $1                       := P#DB22.DBX 0.0 DWORD 80,
           $2                       := P#M 2044.0,
           $3                       := P#DB21.DBX 46.0 DWORD 80);
M013: NOP   0;
      A     L 0.1;
      JNB   M014;
      L     DB22.DBW 8000;
      T     DB21.DBW 384;
M014: NOP   0;
      A     L 0.1;
      JNB   M015;
      L     DB22.DBD 6400;
      T     DB21.DBD 396;
M015: NOP   0;
      A     L 0.1;
      JNB   M016;
      L     DB22.DBD 6404;
      T     DB21.DBD 400;
M016: NOP   0;
      A     L 0.1;
      JNB   M017;
      L     DB22.DBD 6408;
      T     DB21.DBD 404;
M017: NOP   0;
      A     L 0.1;
      JNB   M018;
      L     DB22.DBD 6412;
      T     DB21.DBD 408;
M018: NOP   0;
      A     L 0.1;
      JNB   M019;
      L     DB22.DBW 8040;
      T     DB21.DBW 6;
M019: NOP   0;
      A     L 0.1;
      JNB   M020;
      L     DB22.DBW 8042;
      T     DB21.DBW 8;
M020: NOP   0;
      A     L 0.1;
      JNB   M021;
      L     DB22.DBB 8840;
      T     DB21.DBB 476;
M021: NOP   0;
      A     L 0.0;
      A(;
      L     DB20.DBW 62;
      L     2;
      ==I;
      );
      =     L 0.1;
      A     L 0.1;
      JNB   M022;
      CALL  SFC 20 (
           $1                       := P#DB22.DBX 320.0 DWORD 80,
           $2                       := P#M 2044.0,
           $3                       := P#DB21.DBX 46.0 DWORD 80);
M022: NOP   0;
      A     L 0.1;
      JNB   M023;
      L     DB22.DBW 8002;
      T     DB21.DBW 384;
M023: NOP   0;
      A     L 0.1;
      JNB   M024;
      L     DB22.DBD 6480;
      T     DB21.DBD 396;
M024: NOP   0;
      A     L 0.1;
      JNB   M025;
      L     DB22.DBD 6484;
      T     DB21.DBD 400;
M025: NOP   0;
      A     L 0.1;
      JNB   M026;
      L     DB22.DBD 6488;
      T     DB21.DBD 404;
M026: NOP   0;
      A     L 0.1;
      JNB   M027;
      L     DB22.DBD 6492;
      T     DB21.DBD 408;
M027: NOP   0;
      A     L 0.1;
      JNB   M028;
      L     DB22.DBW 8080;
      T     DB21.DBW 6;
M028: NOP   0;
      A     L 0.1;
      JNB   M029;
      L     DB22.DBW 8082;
      T     DB21.DBW 8;
M029: NOP   0;
      A     L 0.1;
      JNB   M030;
      L     DB22.DBB 8841;
      T     DB21.DBB 476;
M030: NOP   0;
      A     L 0.0;
      A(;
      L     DB20.DBW 62;
      L     3;
      ==I;
      );
      =     L 0.1;
      A     L 0.1;
      JNB   M031;
      CALL  SFC 20 (
           $1                       := P#DB22.DBX 640.0 DWORD 80,
           $2                       := P#M 2044.0,
           $3                       := P#DB21.DBX 46.0 DWORD 80);
M031: NOP   0;
      A     L 0.1;
      JNB   M032;
      L     DB22.DBW 8004;
      T     DB21.DBW 384;
M032: NOP   0;
      A     L 0.1;
      JNB   M033;
      L     DB22.DBD 6560;
      T     DB21.DBD 396;
M033: NOP   0;
      A     L 0.1;
      JNB   M034;
      L     DB22.DBD 6564;
      T     DB21.DBD 400;
M034: NOP   0;
      A     L 0.1;
      JNB   M035;
      L     DB22.DBD 6568;
      T     DB21.DBD 404;
M035: NOP   0;
      A     L 0.1;
      JNB   M036;
      L     DB22.DBD 6572;
      T     DB21.DBD 408;
M036: NOP   0;
      A     L 0.1;
      JNB   M037;
      L     DB22.DBW 8120;
      T     DB21.DBW 6;
M037: NOP   0;
      A     L 0.1;
      JNB   M038;
      L     DB22.DBW 8122;
      T     DB21.DBW 8;
M038: NOP   0;
      A     L 0.1;
      JNB   M039;
      L     DB22.DBB 8842;
      T     DB21.DBB 476;
M039: NOP   0;
      A     L 0.0;
      A(;
      L     DB20.DBW 62;
      L     4;
      ==I;
      );
      =     L 0.1;
      A     L 0.1;
      JNB   M040;
      CALL  SFC 20 (
           $1                       := P#DB22.DBX 960.0 DWORD 80,
           $2                       := P#M 2044.0,
           $3                       := P#DB21.DBX 46.0 DWORD 80);
M040: NOP   0;
      A     L 0.1;
      JNB   M041;
      L     DB22.DBW 8006;
      T     DB21.DBW 384;
M041: NOP   0;
      A     L 0.1;
      JNB   M042;
      L     DB22.DBD 6640;
      T     DB21.DBD 396;
M042: NOP   0;
      A     L 0.1;
      JNB   M043;
      L     DB22.DBD 6644;
      T     DB21.DBD 400;
M043: NOP   0;
      A     L 0.1;
      JNB   M044;
      L     DB22.DBD 6648;
      T     DB21.DBD 404;
M044: NOP   0;
      A     L 0.1;
      JNB   M045;
      L     DB22.DBD 6652;
      T     DB21.DBD 408;
M045: NOP   0;
      A     L 0.1;
      JNB   M046;
      L     DB22.DBW 8160;
      T     DB21.DBW 6;
M046: NOP   0;
      A     L 0.1;
      JNB   M047;
      L     DB22.DBW 8162;
      T     DB21.DBW 8;
M047: NOP   0;
      A     L 0.1;
      JNB   M048;
      L     DB22.DBB 8843;
      T     DB21.DBB 476;
M048: NOP   0;
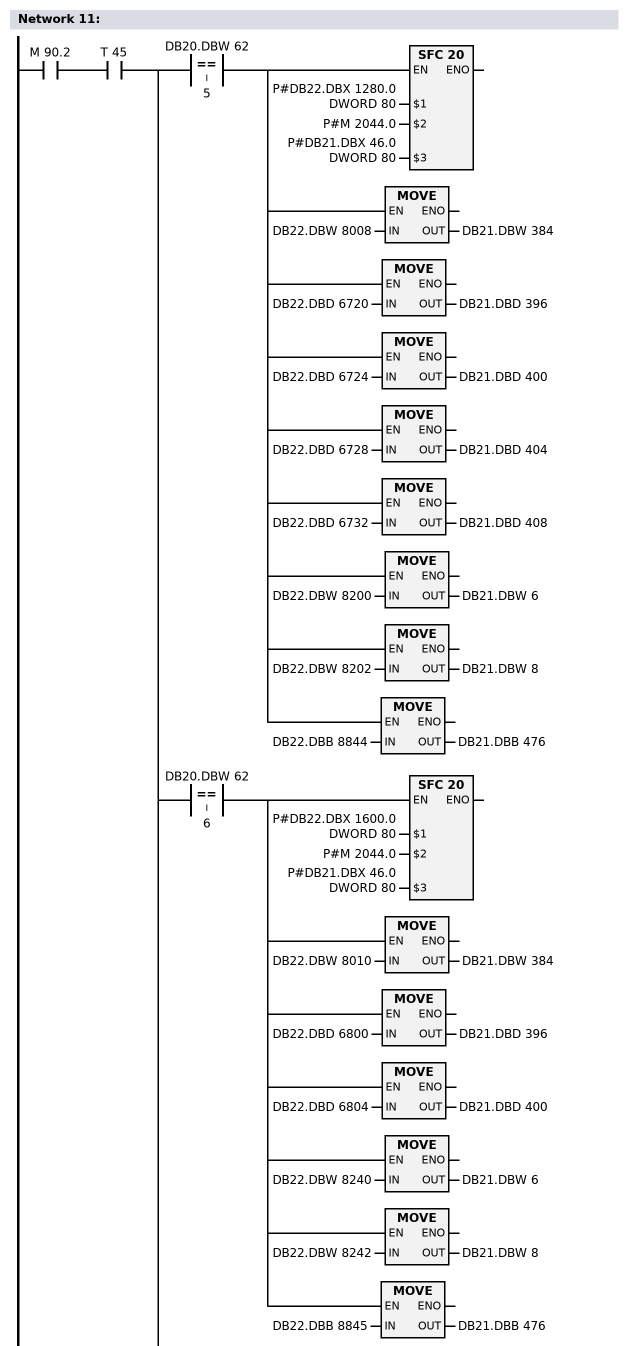
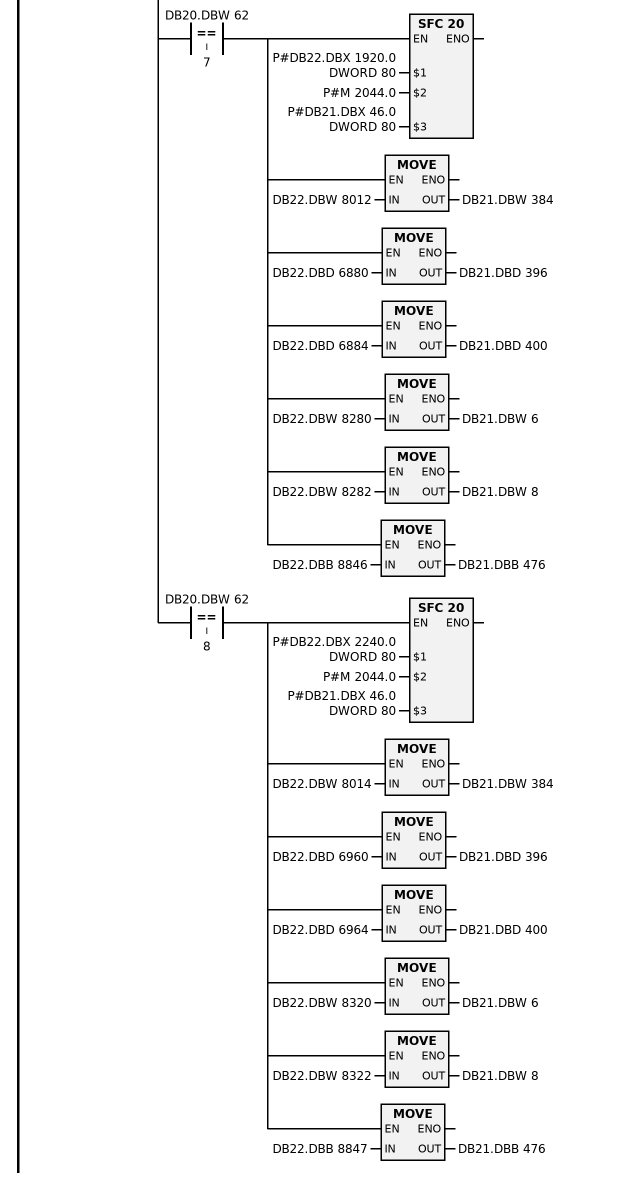
NETWORK
TITLE =
      A     M 90.2;
      A     T 45;
      =     L 0.0;
      A     L 0.0;
      A(;
      L     DB20.DBW 62;
      L     5;
      ==I;
      );
      =     L 0.1;
      A     L 0.1;
      JNB   M049;
      CALL  SFC 20 (
           $1                       := P#DB22.DBX 1280.0 DWORD 80,
           $2                       := P#M 2044.0,
           $3                       := P#DB21.DBX 46.0 DWORD 80);
M049: NOP   0;
      A     L 0.1;
      JNB   M050;
      L     DB22.DBW 8008;
      T     DB21.DBW 384;
M050: NOP   0;
      A     L 0.1;
      JNB   M051;
      L     DB22.DBD 6720;
      T     DB21.DBD 396;
M051: NOP   0;
      A     L 0.1;
      JNB   M052;
      L     DB22.DBD 6724;
      T     DB21.DBD 400;
M052: NOP   0;
      A     L 0.1;
      JNB   M053;
      L     DB22.DBD 6728;
      T     DB21.DBD 404;
M053: NOP   0;
      A     L 0.1;
      JNB   M054;
      L     DB22.DBD 6732;
      T     DB21.DBD 408;
M054: NOP   0;
      A     L 0.1;
      JNB   M055;
      L     DB22.DBW 8200;
      T     DB21.DBW 6;
M055: NOP   0;
      A     L 0.1;
      JNB   M056;
      L     DB22.DBW 8202;
      T     DB21.DBW 8;
M056: NOP   0;
      A     L 0.1;
      JNB   M057;
      L     DB22.DBB 8844;
      T     DB21.DBB 476;
M057: NOP   0;
      A     L 0.0;
      A(;
      L     DB20.DBW 62;
      L     6;
      ==I;
      );
      =     L 0.1;
      A     L 0.1;
      JNB   M058;
      CALL  SFC 20 (
           $1                       := P#DB22.DBX 1600.0 DWORD 80,
           $2                       := P#M 2044.0,
           $3                       := P#DB21.DBX 46.0 DWORD 80);
M058: NOP   0;
      A     L 0.1;
      JNB   M059;
      L     DB22.DBW 8010;
      T     DB21.DBW 384;
M059: NOP   0;
      A     L 0.1;
      JNB   M060;
      L     DB22.DBD 6800;
      T     DB21.DBD 396;
M060: NOP   0;
      A     L 0.1;
      JNB   M061;
      L     DB22.DBD 6804;
      T     DB21.DBD 400;
M061: NOP   0;
      A     L 0.1;
      JNB   M062;
      L     DB22.DBW 8240;
      T     DB21.DBW 6;
M062: NOP   0;
      A     L 0.1;
      JNB   M063;
      L     DB22.DBW 8242;
      T     DB21.DBW 8;
M063: NOP   0;
      A     L 0.1;
      JNB   M064;
      L     DB22.DBB 8845;
      T     DB21.DBB 476;
M064: NOP   0;
      A     L 0.0;
      A(;
      L     DB20.DBW 62;
      L     7;
      ==I;
      );
      =     L 0.1;
      A     L 0.1;
      JNB   M065;
      CALL  SFC 20 (
           $1                       := P#DB22.DBX 1920.0 DWORD 80,
           $2                       := P#M 2044.0,
           $3                       := P#DB21.DBX 46.0 DWORD 80);
M065: NOP   0;
      A     L 0.1;
      JNB   M066;
      L     DB22.DBW 8012;
      T     DB21.DBW 384;
M066: NOP   0;
      A     L 0.1;
      JNB   M067;
      L     DB22.DBD 6880;
      T     DB21.DBD 396;
M067: NOP   0;
      A     L 0.1;
      JNB   M068;
      L     DB22.DBD 6884;
      T     DB21.DBD 400;
M068: NOP   0;
      A     L 0.1;
      JNB   M069;
      L     DB22.DBW 8280;
      T     DB21.DBW 6;
M069: NOP   0;
      A     L 0.1;
      JNB   M070;
      L     DB22.DBW 8282;
      T     DB21.DBW 8;
M070: NOP   0;
      A     L 0.1;
      JNB   M071;
      L     DB22.DBB 8846;
      T     DB21.DBB 476;
M071: NOP   0;
      A     L 0.0;
      A(;
      L     DB20.DBW 62;
      L     8;
      ==I;
      );
      =     L 0.1;
      A     L 0.1;
      JNB   M072;
      CALL  SFC 20 (
           $1                       := P#DB22.DBX 2240.0 DWORD 80,
           $2                       := P#M 2044.0,
           $3                       := P#DB21.DBX 46.0 DWORD 80);
M072: NOP   0;
      A     L 0.1;
      JNB   M073;
      L     DB22.DBW 8014;
      T     DB21.DBW 384;
M073: NOP   0;
      A     L 0.1;
      JNB   M074;
      L     DB22.DBD 6960;
      T     DB21.DBD 396;
M074: NOP   0;
      A     L 0.1;
      JNB   M075;
      L     DB22.DBD 6964;
      T     DB21.DBD 400;
M075: NOP   0;
      A     L 0.1;
      JNB   M076;
      L     DB22.DBW 8320;
      T     DB21.DBW 6;
M076: NOP   0;
      A     L 0.1;
      JNB   M077;
      L     DB22.DBW 8322;
      T     DB21.DBW 8;
M077: NOP   0;
      A     L 0.1;
      JNB   M078;
      L     DB22.DBB 8847;
      T     DB21.DBB 476;
M078: NOP   0;
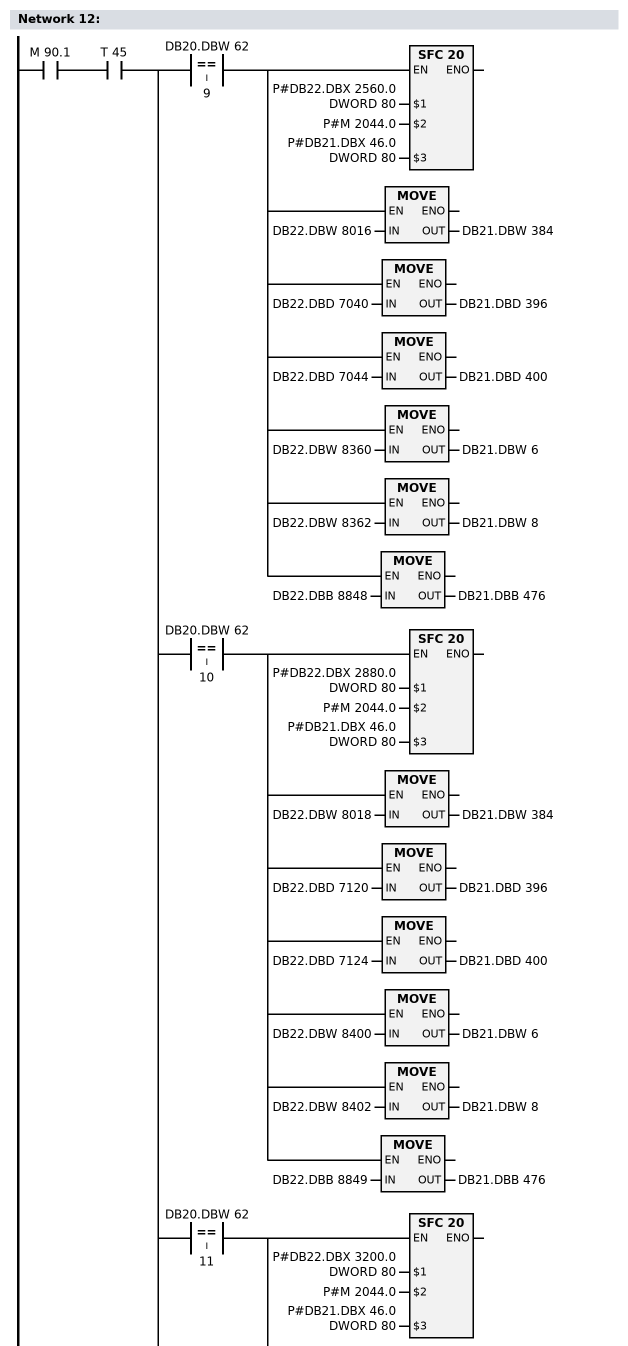
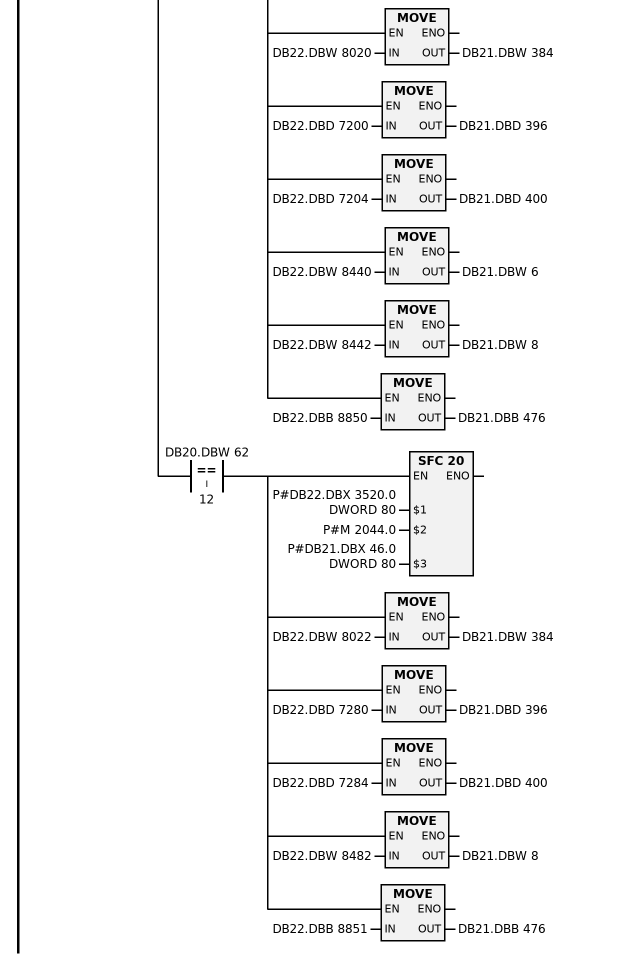
NETWORK
TITLE =
      A     M 90.1;
      A     T 45;
      =     L 0.0;
      A     L 0.0;
      A(;
      L     DB20.DBW 62;
      L     9;
      ==I;
      );
      =     L 0.1;
      A     L 0.1;
      JNB   M079;
      CALL  SFC 20 (
           $1                       := P#DB22.DBX 2560.0 DWORD 80,
           $2                       := P#M 2044.0,
           $3                       := P#DB21.DBX 46.0 DWORD 80);
M079: NOP   0;
      A     L 0.1;
      JNB   M080;
      L     DB22.DBW 8016;
      T     DB21.DBW 384;
M080: NOP   0;
      A     L 0.1;
      JNB   M081;
      L     DB22.DBD 7040;
      T     DB21.DBD 396;
M081: NOP   0;
      A     L 0.1;
      JNB   M082;
      L     DB22.DBD 7044;
      T     DB21.DBD 400;
M082: NOP   0;
      A     L 0.1;
      JNB   M083;
      L     DB22.DBW 8360;
      T     DB21.DBW 6;
M083: NOP   0;
      A     L 0.1;
      JNB   M084;
      L     DB22.DBW 8362;
      T     DB21.DBW 8;
M084: NOP   0;
      A     L 0.1;
      JNB   M085;
      L     DB22.DBB 8848;
      T     DB21.DBB 476;
M085: NOP   0;
      A     L 0.0;
      A(;
      L     DB20.DBW 62;
      L     10;
      ==I;
      );
      =     L 0.1;
      A     L 0.1;
      JNB   M086;
      CALL  SFC 20 (
           $1                       := P#DB22.DBX 2880.0 DWORD 80,
           $2                       := P#M 2044.0,
           $3                       := P#DB21.DBX 46.0 DWORD 80);
M086: NOP   0;
      A     L 0.1;
      JNB   M087;
      L     DB22.DBW 8018;
      T     DB21.DBW 384;
M087: NOP   0;
      A     L 0.1;
      JNB   M088;
      L     DB22.DBD 7120;
      T     DB21.DBD 396;
M088: NOP   0;
      A     L 0.1;
      JNB   M089;
      L     DB22.DBD 7124;
      T     DB21.DBD 400;
M089: NOP   0;
      A     L 0.1;
      JNB   M090;
      L     DB22.DBW 8400;
      T     DB21.DBW 6;
M090: NOP   0;
      A     L 0.1;
      JNB   M091;
      L     DB22.DBW 8402;
      T     DB21.DBW 8;
M091: NOP   0;
      A     L 0.1;
      JNB   M092;
      L     DB22.DBB 8849;
      T     DB21.DBB 476;
M092: NOP   0;
      A     L 0.0;
      A(;
      L     DB20.DBW 62;
      L     11;
      ==I;
      );
      =     L 0.1;
      A     L 0.1;
      JNB   M093;
      CALL  SFC 20 (
           $1                       := P#DB22.DBX 3200.0 DWORD 80,
           $2                       := P#M 2044.0,
           $3                       := P#DB21.DBX 46.0 DWORD 80);
M093: NOP   0;
      A     L 0.1;
      JNB   M094;
      L     DB22.DBW 8020;
      T     DB21.DBW 384;
M094: NOP   0;
      A     L 0.1;
      JNB   M095;
      L     DB22.DBD 7200;
      T     DB21.DBD 396;
M095: NOP   0;
      A     L 0.1;
      JNB   M096;
      L     DB22.DBD 7204;
      T     DB21.DBD 400;
M096: NOP   0;
      A     L 0.1;
      JNB   M097;
      L     DB22.DBW 8440;
      T     DB21.DBW 6;
M097: NOP   0;
      A     L 0.1;
      JNB   M098;
      L     DB22.DBW 8442;
      T     DB21.DBW 8;
M098: NOP   0;
      A     L 0.1;
      JNB   M099;
      L     DB22.DBB 8850;
      T     DB21.DBB 476;
M099: NOP   0;
      A     L 0.0;
      A(;
      L     DB20.DBW 62;
      L     12;
      ==I;
      );
      =     L 0.1;
      A     L 0.1;
      JNB   M100;
      CALL  SFC 20 (
           $1                       := P#DB22.DBX 3520.0 DWORD 80,
           $2                       := P#M 2044.0,
           $3                       := P#DB21.DBX 46.0 DWORD 80);
M100: NOP   0;
      A     L 0.1;
      JNB   M101;
      L     DB22.DBW 8022;
      T     DB21.DBW 384;
M101: NOP   0;
      A     L 0.1;
      JNB   M102;
      L     DB22.DBD 7280;
      T     DB21.DBD 396;
M102: NOP   0;
      A     L 0.1;
      JNB   M103;
      L     DB22.DBD 7284;
      T     DB21.DBD 400;
M103: NOP   0;
      A     L 0.1;
      JNB   M104;
      L     DB22.DBW 8482;
      T     DB21.DBW 8;
M104: NOP   0;
      A     L 0.1;
      JNB   M105;
      L     DB22.DBB 8851;
      T     DB21.DBB 476;
M105: NOP   0;
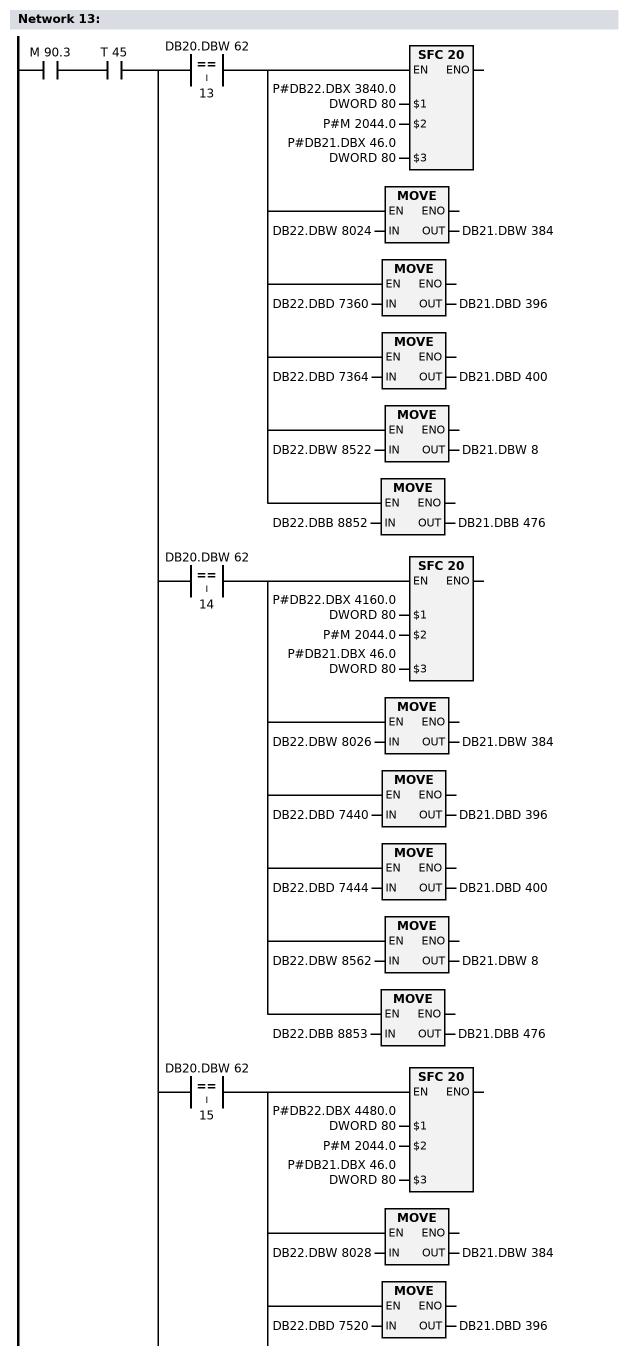
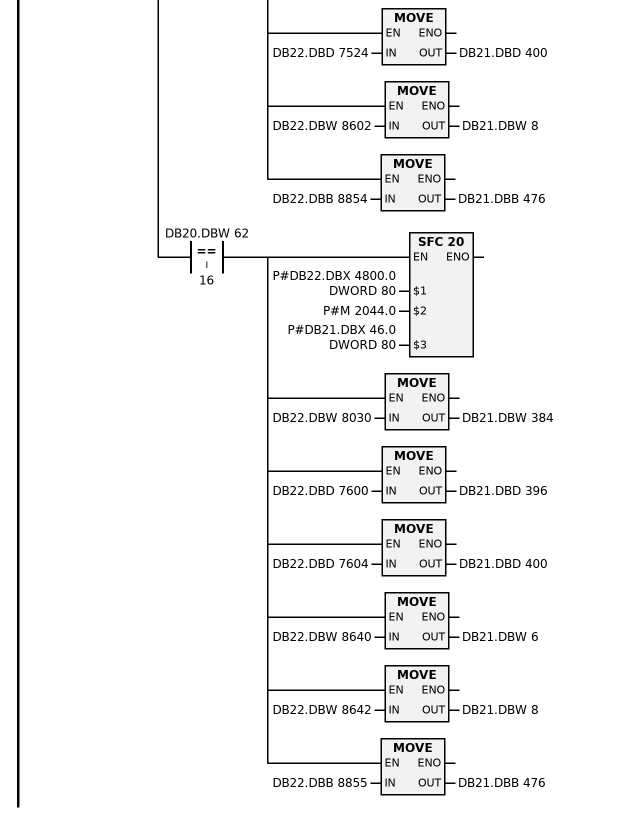
NETWORK
TITLE =
      A     M 90.3;
      A     T 45;
      =     L 0.0;
      A     L 0.0;
      A(;
      L     DB20.DBW 62;
      L     13;
      ==I;
      );
      =     L 0.1;
      A     L 0.1;
      JNB   M106;
      CALL  SFC 20 (
           $1                       := P#DB22.DBX 3840.0 DWORD 80,
           $2                       := P#M 2044.0,
           $3                       := P#DB21.DBX 46.0 DWORD 80);
M106: NOP   0;
      A     L 0.1;
      JNB   M107;
      L     DB22.DBW 8024;
      T     DB21.DBW 384;
M107: NOP   0;
      A     L 0.1;
      JNB   M108;
      L     DB22.DBD 7360;
      T     DB21.DBD 396;
M108: NOP   0;
      A     L 0.1;
      JNB   M109;
      L     DB22.DBD 7364;
      T     DB21.DBD 400;
M109: NOP   0;
      A     L 0.1;
      JNB   M110;
      L     DB22.DBW 8522;
      T     DB21.DBW 8;
M110: NOP   0;
      A     L 0.1;
      JNB   M111;
      L     DB22.DBB 8852;
      T     DB21.DBB 476;
M111: NOP   0;
      A     L 0.0;
      A(;
      L     DB20.DBW 62;
      L     14;
      ==I;
      );
      =     L 0.1;
      A     L 0.1;
      JNB   M112;
      CALL  SFC 20 (
           $1                       := P#DB22.DBX 4160.0 DWORD 80,
           $2                       := P#M 2044.0,
           $3                       := P#DB21.DBX 46.0 DWORD 80);
M112: NOP   0;
      A     L 0.1;
      JNB   M113;
      L     DB22.DBW 8026;
      T     DB21.DBW 384;
M113: NOP   0;
      A     L 0.1;
      JNB   M114;
      L     DB22.DBD 7440;
      T     DB21.DBD 396;
M114: NOP   0;
      A     L 0.1;
      JNB   M115;
      L     DB22.DBD 7444;
      T     DB21.DBD 400;
M115: NOP   0;
      A     L 0.1;
      JNB   M116;
      L     DB22.DBW 8562;
      T     DB21.DBW 8;
M116: NOP   0;
      A     L 0.1;
      JNB   M117;
      L     DB22.DBB 8853;
      T     DB21.DBB 476;
M117: NOP   0;
      A     L 0.0;
      A(;
      L     DB20.DBW 62;
      L     15;
      ==I;
      );
      =     L 0.1;
      A     L 0.1;
      JNB   M118;
      CALL  SFC 20 (
           $1                       := P#DB22.DBX 4480.0 DWORD 80,
           $2                       := P#M 2044.0,
           $3                       := P#DB21.DBX 46.0 DWORD 80);
M118: NOP   0;
      A     L 0.1;
      JNB   M119;
      L     DB22.DBW 8028;
      T     DB21.DBW 384;
M119: NOP   0;
      A     L 0.1;
      JNB   M120;
      L     DB22.DBD 7520;
      T     DB21.DBD 396;
M120: NOP   0;
      A     L 0.1;
      JNB   M121;
      L     DB22.DBD 7524;
      T     DB21.DBD 400;
M121: NOP   0;
      A     L 0.1;
      JNB   M122;
      L     DB22.DBW 8602;
      T     DB21.DBW 8;
M122: NOP   0;
      A     L 0.1;
      JNB   M123;
      L     DB22.DBB 8854;
      T     DB21.DBB 476;
M123: NOP   0;
      A     L 0.0;
      A(;
      L     DB20.DBW 62;
      L     16;
      ==I;
      );
      =     L 0.1;
      A     L 0.1;
      JNB   M124;
      CALL  SFC 20 (
           $1                       := P#DB22.DBX 4800.0 DWORD 80,
           $2                       := P#M 2044.0,
           $3                       := P#DB21.DBX 46.0 DWORD 80);
M124: NOP   0;
      A     L 0.1;
      JNB   M125;
      L     DB22.DBW 8030;
      T     DB21.DBW 384;
M125: NOP   0;
      A     L 0.1;
      JNB   M126;
      L     DB22.DBD 7600;
      T     DB21.DBD 396;
M126: NOP   0;
      A     L 0.1;
      JNB   M127;
      L     DB22.DBD 7604;
      T     DB21.DBD 400;
M127: NOP   0;
      A     L 0.1;
      JNB   M128;
      L     DB22.DBW 8640;
      T     DB21.DBW 6;
M128: NOP   0;
      A     L 0.1;
      JNB   M129;
      L     DB22.DBW 8642;
      T     DB21.DBW 8;
M129: NOP   0;
      A     L 0.1;
      JNB   M130;
      L     DB22.DBB 8855;
      T     DB21.DBB 476;
M130: NOP   0;
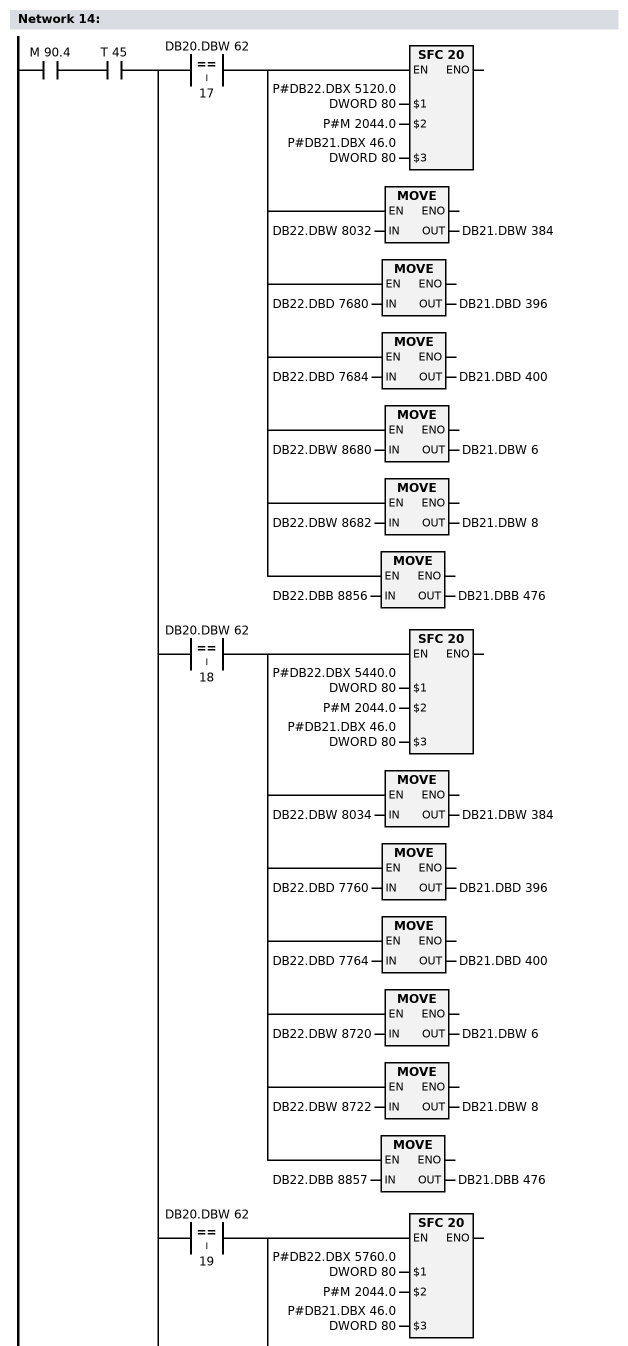
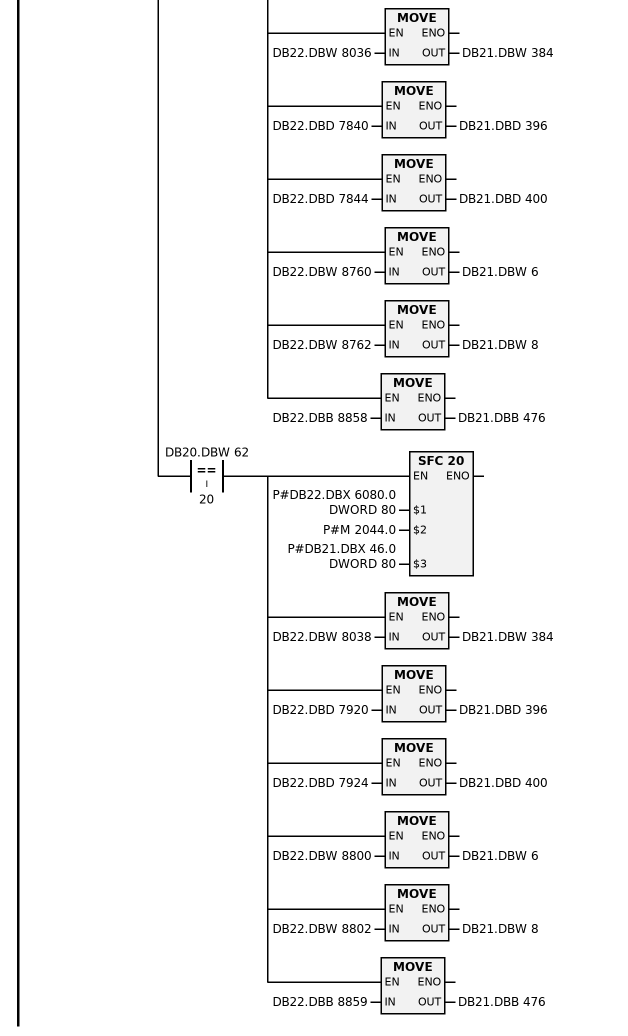
NETWORK
TITLE =
      A     M 90.4;
      A     T 45;
      =     L 0.0;
      A     L 0.0;
      A(;
      L     DB20.DBW 62;
      L     17;
      ==I;
      );
      =     L 0.1;
      A     L 0.1;
      JNB   M131;
      CALL  SFC 20 (
           $1                       := P#DB22.DBX 5120.0 DWORD 80,
           $2                       := P#M 2044.0,
           $3                       := P#DB21.DBX 46.0 DWORD 80);
M131: NOP   0;
      A     L 0.1;
      JNB   M132;
      L     DB22.DBW 8032;
      T     DB21.DBW 384;
M132: NOP   0;
      A     L 0.1;
      JNB   M133;
      L     DB22.DBD 7680;
      T     DB21.DBD 396;
M133: NOP   0;
      A     L 0.1;
      JNB   M134;
      L     DB22.DBD 7684;
      T     DB21.DBD 400;
M134: NOP   0;
      A     L 0.1;
      JNB   M135;
      L     DB22.DBW 8680;
      T     DB21.DBW 6;
M135: NOP   0;
      A     L 0.1;
      JNB   M136;
      L     DB22.DBW 8682;
      T     DB21.DBW 8;
M136: NOP   0;
      A     L 0.1;
      JNB   M137;
      L     DB22.DBB 8856;
      T     DB21.DBB 476;
M137: NOP   0;
      A     L 0.0;
      A(;
      L     DB20.DBW 62;
      L     18;
      ==I;
      );
      =     L 0.1;
      A     L 0.1;
      JNB   M138;
      CALL  SFC 20 (
           $1                       := P#DB22.DBX 5440.0 DWORD 80,
           $2                       := P#M 2044.0,
           $3                       := P#DB21.DBX 46.0 DWORD 80);
M138: NOP   0;
      A     L 0.1;
      JNB   M139;
      L     DB22.DBW 8034;
      T     DB21.DBW 384;
M139: NOP   0;
      A     L 0.1;
      JNB   M140;
      L     DB22.DBD 7760;
      T     DB21.DBD 396;
M140: NOP   0;
      A     L 0.1;
      JNB   M141;
      L     DB22.DBD 7764;
      T     DB21.DBD 400;
M141: NOP   0;
      A     L 0.1;
      JNB   M142;
      L     DB22.DBW 8720;
      T     DB21.DBW 6;
M142: NOP   0;
      A     L 0.1;
      JNB   M143;
      L     DB22.DBW 8722;
      T     DB21.DBW 8;
M143: NOP   0;
      A     L 0.1;
      JNB   M144;
      L     DB22.DBB 8857;
      T     DB21.DBB 476;
M144: NOP   0;
      A     L 0.0;
      A(;
      L     DB20.DBW 62;
      L     19;
      ==I;
      );
      =     L 0.1;
      A     L 0.1;
      JNB   M145;
      CALL  SFC 20 (
           $1                       := P#DB22.DBX 5760.0 DWORD 80,
           $2                       := P#M 2044.0,
           $3                       := P#DB21.DBX 46.0 DWORD 80);
M145: NOP   0;
      A     L 0.1;
      JNB   M146;
      L     DB22.DBW 8036;
      T     DB21.DBW 384;
M146: NOP   0;
      A     L 0.1;
      JNB   M147;
      L     DB22.DBD 7840;
      T     DB21.DBD 396;
M147: NOP   0;
      A     L 0.1;
      JNB   M148;
      L     DB22.DBD 7844;
      T     DB21.DBD 400;
M148: NOP   0;
      A     L 0.1;
      JNB   M149;
      L     DB22.DBW 8760;
      T     DB21.DBW 6;
M149: NOP   0;
      A     L 0.1;
      JNB   M150;
      L     DB22.DBW 8762;
      T     DB21.DBW 8;
M150: NOP   0;
      A     L 0.1;
      JNB   M151;
      L     DB22.DBB 8858;
      T     DB21.DBB 476;
M151: NOP   0;
      A     L 0.0;
      A(;
      L     DB20.DBW 62;
      L     20;
      ==I;
      );
      =     L 0.1;
      A     L 0.1;
      JNB   M152;
      CALL  SFC 20 (
           $1                       := P#DB22.DBX 6080.0 DWORD 80,
           $2                       := P#M 2044.0,
           $3                       := P#DB21.DBX 46.0 DWORD 80);
M152: NOP   0;
      A     L 0.1;
      JNB   M153;
      L     DB22.DBW 8038;
      T     DB21.DBW 384;
M153: NOP   0;
      A     L 0.1;
      JNB   M154;
      L     DB22.DBD 7920;
      T     DB21.DBD 396;
M154: NOP   0;
      A     L 0.1;
      JNB   M155;
      L     DB22.DBD 7924;
      T     DB21.DBD 400;
M155: NOP   0;
      A     L 0.1;
      JNB   M156;
      L     DB22.DBW 8800;
      T     DB21.DBW 6;
M156: NOP   0;
      A     L 0.1;
      JNB   M157;
      L     DB22.DBW 8802;
      T     DB21.DBW 8;
M157: NOP   0;
      A     L 0.1;
      JNB   M158;
      L     DB22.DBB 8859;
      T     DB21.DBB 476;
M158: NOP   0;
END_FUNCTION

FUNCTION FC 52 : VOID
VERSION : 0.1
BEGIN
// (block stored without names or comments; labels and parameter names are numbered)
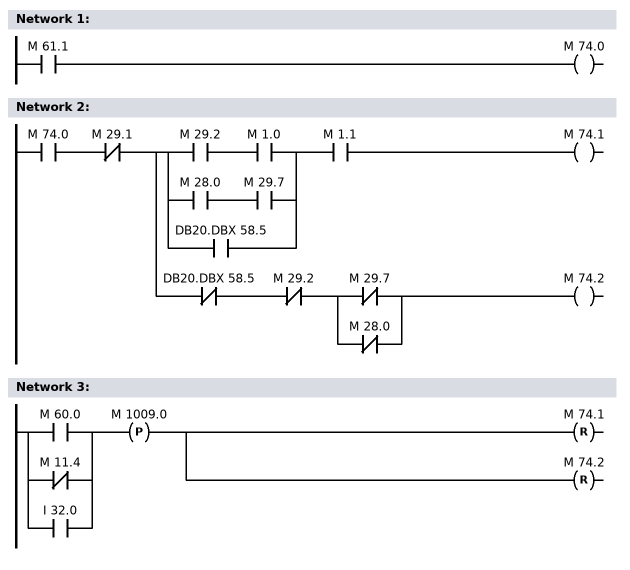
NETWORK
TITLE =
      A     M 61.1;
      =     M 74.0;
NETWORK
TITLE =
      A     M 74.0;
      AN    M 29.1;
      =     L 0.0;
      A     L 0.0;
      A(;
      A     M 29.2;
      A     M 1.0;
      O;
      A     M 28.0;
      A     M 29.7;
      O     DB20.DBX 58.5;
      );
      A     M 1.1;
      =     M 74.1;
      A     L 0.0;
      AN    DB20.DBX 58.5;
      AN    M 29.2;
      A(;
      ON    M 29.7;
      ON    M 28.0;
      );
      =     M 74.2;
NETWORK
TITLE =
      A(;
      O     M 60.0;
      ON    M 11.4;
      O     I 32.0;
      );
      FP    M 1009.0;
      R     M 74.1;
      R     M 74.2;
END_FUNCTION

FUNCTION FC 53 : VOID
VERSION : 0.1
BEGIN
// (block stored without names or comments; labels and parameter names are numbered)
NETWORK
TITLE =
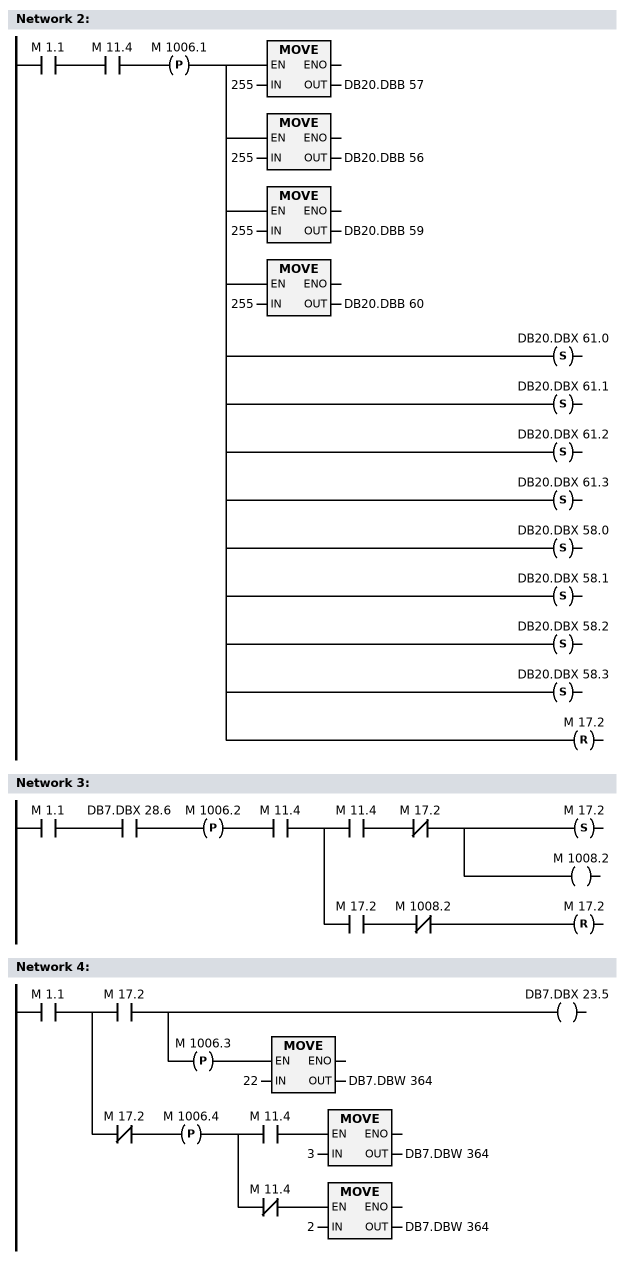
NETWORK
TITLE =
      A     M 1.1;
      A     M 11.4;
      FP    M 1006.1;
      =     L 0.0;
      A     L 0.0;
      JNB   M001;
      L     255;
      T     DB20.DBB 57;
M001: NOP   0;
      A     L 0.0;
      JNB   M002;
      L     255;
      T     DB20.DBB 56;
M002: NOP   0;
      A     L 0.0;
      JNB   M003;
      L     255;
      T     DB20.DBB 59;
M003: NOP   0;
      A     L 0.0;
      JNB   M004;
      L     255;
      T     DB20.DBB 60;
M004: NOP   0;
      A     L 0.0;
      BLD   102;
      S     DB20.DBX 61.0;
      A     L 0.0;
      BLD   102;
      S     DB20.DBX 61.1;
      A     L 0.0;
      BLD   102;
      S     DB20.DBX 61.2;
      A     L 0.0;
      BLD   102;
      S     DB20.DBX 61.3;
      A     L 0.0;
      BLD   102;
      S     DB20.DBX 58.0;
      A     L 0.0;
      BLD   102;
      S     DB20.DBX 58.1;
      A     L 0.0;
      BLD   102;
      S     DB20.DBX 58.2;
      A     L 0.0;
      BLD   102;
      S     DB20.DBX 58.3;
      A     L 0.0;
      BLD   102;
      R     M 17.2;
NETWORK
TITLE =
      A     M 1.1;
      A     DB7.DBX 28.6;
      FP    M 1006.2;
      A     M 11.4;
      =     L 0.0;
      A     L 0.0;
      A     M 11.4;
      AN    M 17.2;
      S     M 17.2;
      =     M 1008.2;
      A     L 0.0;
      A     M 17.2;
      AN    M 1008.2;
      R     M 17.2;
NETWORK
TITLE =
      A     M 1.1;
      =     L 0.0;
      A     L 0.0;
      A     M 17.2;
      =     L 0.1;
      A     L 0.1;
      BLD   102;
      =     DB7.DBX 23.5;
      A     L 0.1;
      FP    M 1006.3;
      JNB   M005;
      L     22;
      T     DB7.DBW 364;
M005: NOP   0;
      A     L 0.0;
      AN    M 17.2;
      FP    M 1006.4;
      =     L 0.1;
      A     L 0.1;
      A     M 11.4;
      JNB   M006;
      L     3;
      T     DB7.DBW 364;
M006: NOP   0;
      A     L 0.1;
      AN    M 11.4;
      JNB   M007;
      L     2;
      T     DB7.DBW 364;
M007: NOP   0;
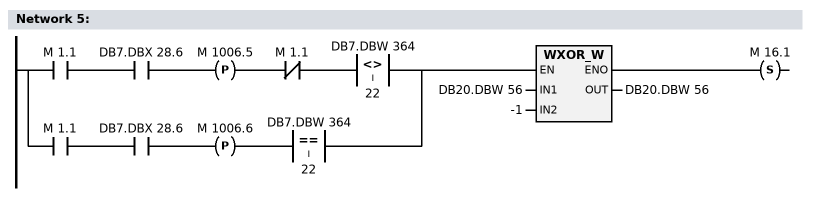
NETWORK
TITLE =
      A(;
      A     M 1.1;
      A     DB7.DBX 28.6;
      FP    M 1006.5;
      AN    M 1.1;
      A(;
      L     DB7.DBW 364;
      L     22;
      <>I;
      );
      O(;
      A     M 1.1;
      A     DB7.DBX 28.6;
      FP    M 1006.6;
      A(;
      L     DB7.DBW 364;
      L     22;
      ==I;
      );
      );
      );
      JNB   M008;
      L     DB20.DBW 56;
      L     -1;
      XOW;
      T     DB20.DBW 56;
      SET;
      SAVE;
      CLR;
M008: A     BR;
      S     M 16.1;
